     bHomed         :BOOL; 
     Pos_Done       :BOOL;   //定位完成
     Home_Alm      :BOOL;  //回零超时报警
     Pos_Alm         :BOOL; //定位超时报警



END_STRUCT
END_TYPE

// ---- P2DUTs/01_AxisCO_Ntrol/ST_JXCE.TcDUT
TYPE ST_JXCE :
STRUCT
      out_Control             AT  %Q*  :     UINT;  // 电机控制
      out_Function            AT  %Q*  :    UINT;  // 电机功能
      out_Start                 AT  %Q*  :   USINT;  // 电机启动定位
      out_Mode               AT  %Q*  :   USINT;  // 电机定位模式
      out_Cmd_Vel           AT  %Q*  :    UINT;  // 电机命令速度
      out_Cmd_Pos           AT  %Q*  :   DINT;  // 电机命令位置
      out_Cmd_Acc           AT  %Q*  :   UINT;  // 电机命令加速度
      out_Cmd_Dec          AT  %Q*  :    UINT;  // 电机命令减速度

      in_Status               AT  %I*  :     UINT;  // 电机状态
      in_Flag                 AT  %I*  :     UINT;  // 电机标志位
      in_Act_Pos              AT  %I*  :     DINT;  // 电机反馈位置
      in_Act_Vel             AT  %I*  :     UINT;  // 电机反馈速度
   
     in_Latest_Alm          AT  %I*  :     USINT;  // 电机最新报警

END_STRUCT
END_TYPE

// ---- P2DUTs/01_AxisCO_Ntrol/ST_SetpMotor.TcDUT
TYPE ST_SetpMotor :
STRUCT
	bJog_Up			:BOOL;		
	bJog_Down			:BOOL;	 
	bHome			:BOOL;	 
	bGoWorkPos			:BOOL;	 
	bLeaveWorkPos			:BOOL;	 
	HomeDone    :BOOL;  
	WorkPosDone :BOOL;
	
	
	
	biSensor  :BOOL;   //对射关电
	biUpSensor  :BOOL;   
	biRefSensor  :BOOL;   
	biMiddle2Sensor  :BOOL;   //步进中位感应 无用
	biDownSensor  :BOOL;  
	biBoxSensor  :BOOL;   //料盒到位感应
	bHave			:BOOL;//有料感应
	
	bo_Up			:BOOL;		
	bo_Down			:BOOL;	    

	bPoleFull: BOOL;  //极片料满

END_STRUCT
END_TYPE

// ---- P2DUTs/01_AxisCO_Ntrol_1/ST_AxisCmd.TcDUT
TYPE ST_AxisCmd :  //轴运动控制相关
STRUCT

   bDynamitcsParSel      :INT:=1;  // 1:NC          2:UserDefine


	bEnable			        :BOOL;				    (*使能*)
	fOverride			    :REAL:=100;			(*MC_power中实际倍率的设定，默认值为100*)
	bEnableFw		        :BOOL:=TRUE;		 (*正向使能*)
	bEnableBw		    :BOOL:=TRUE;	 	(*负向使能*)

	bJog_Fw			    :BOOL;			     	(*正向点动*)
	bJog_Bw			    :BOOL;			    	(*反向点动*)

	bMoveAbs	 	        :BOOL;				    (*运行绝对位置*)
	fPositon_of_Abs	 	:REAL;					(*绝对位置位移*)

	bMoveRel		        :BOOL;				   (*运行当对位置*)
	fPosition_of_Rel	    :REAL;				   (*相对位置位移*)

	bMoveModulo		 :BOOL;				     (*运行模长位置*)
	fPositon_of_Mod	  :REAL;					  (*模长位置位移*)

	bMoveVelo		    :BOOL;				       (*向一个方向持续运行，方向由前面的正向点动或者反向点动设置*)
	bMoveVeloDir	:MC_Direction := MC_Positive_Direction ;	(*速度运动的方向,MC_Negative_Direction*)

	bHome			       :BOOL;						(*启动回参*)

	bSetPos			       :BOOL;						 (*设置轴当前的位置为一个绝对位置*)
    fSetPos				   :REAL:=0;					(*setpos功能块将轴当前的位置设置为这个变量*)

	iGoSetPos              :INT;                     //GO离散点位_INT
    arrbGoSetPos      :ARRAY[0..15]        OF BOOL;  //GO离散点位_布尔数组
	iRealPoint              :INT;                     //离散点位指示_INIT
    arrbRealPoint        :ARRAY[0..15]        OF BOOL;  //离散点位指示_布尔数组

	bHalt			            :BOOL;				(*暂停*)
	bStop			        :BOOL;				(*停止*)
	bGearOut			    :BOOL;				(*解耦*)
	bReset			        :BOOL;				(*复位*)

	hmiJog_Fw			    :BOOL;				//正向点动_BOOL
	hmibJog_Bw		     :BOOL;				//反向点动_BOOL	
	hmiGoSetPos          :INT;              //GO离散点位_INT


//条件
     Home_Condition       :BOOL:=TRUE;//回原点条件
     JogP_Condition       :BOOL:=TRUE;//点动正转条件
     JogN_Condition       :BOOL:=TRUE;//点动反转条件
     GoPoint_Condition    :ARRAY[0..15] OF BOOL;//HMI点动定位条件


//轴到位判断
	Axis_R:REAL:=0.13;//轴到位判断





END_STRUCT
END_TYPE

// ---- P2DUTs/01_AxisCO_Ntrol_1/ST_AxisCtrl.TcDUT
TYPE ST_AxisCtrl :
STRUCT
    Io                        :ST_AxisIo;  (*轴IO信号*)
    Status                  :ST_AxisStatus;  
    Cmd                    :ST_AxisCmd;  
END_STRUCT
END_TYPE

// ---- P2DUTs/01_AxisCO_Ntrol_1/ST_AxisIo.TcDUT
TYPE ST_AxisIo :   //轴IO信号
STRUCT

	biNegLimit	             :BOOL;		            (*负限位触发信号*)
	biPosLimit	             :BOOL;		            (*正限位触发信号*)
	biHomeSwitch	     :BOOL;		         (*原点触发信号*)
    DigitalInputs          AT %I*	:  UDINT;
	
END_STRUCT
END_TYPE

// ---- P2DUTs/01_AxisCO_Ntrol_1/ST_AxisStatus.TcDUT
TYPE ST_AxisStatus :   //轴相关状态
STRUCT

(*status*)
	AxisName		     :STRING(31);		     (*轴名称*)
	AxisID			     :UDINT;		      (*轴在NC中的编号*)
	
    Enabled		         :BOOL;              //使能状态
	Moving              :BOOL;                //轴运行中
	NoMoving          :BOOL;   //轴停止中
    Coupled             :BOOL;   //轴耦合中

	fActPos			     :LREAL;  //轴的当前位置               
	fSetPos			     :LREAL;   //轴的指令位置              
    fModuloActPos		 :REAL;   //轴的当前模长位置             
    fModuloSetPos		 :REAL;      //轴的指令模长位置 
    fActVelo			   :REAL;    //轴的当前速度             
    fSetVelo			   :REAL;    //轴的指令速度
	Homed                :BOOL;        //轴回原点完成         
 
	Error                   :BOOL;//轴报错
	ErrorID                  :UDINT;//轴报错ID号
    WarningDynamitcsPar    :BOOL; //运动参数警告

     ErrorLimitSwitch           :BOOL; //限位报警
	 Errorcomp                   :BOOL; //手自动报警
END_STRUCT
END_TYPE

// ---- P2DUTs/01_AxisCO_Ntrol_1/ST_Axis_Par.TcDUT
TYPE ST_Axis_Par ://轴参数
STRUCT
    bLimitSwitchEn          :BOOL;//限位保护开启


	fVelocity_of_Abs	 :REAL:=5;				
	fVelocity_of_Mod	 :REAL:=5;				
	fVelocity_of_Rel	 :REAL:=5;				
	fVelocity_of_Velo	 :REAL:=5;				
	fVelocity_of_Jog	 :REAL:=10;			
	fInchingDistance	 :REAL:=5;				

	arrTargetPoint : ARRAY [0..15] OF REAL ;
	//fMaxVelocity:        REAL:=0;	
    fTagatTime                                 :REAL:=0.5;//S
    fConVelPercentage                      :REAL:=0.8;//S
    fMaxAccDec                              :LREAL:=40000;//最大加速度
    fMaxVel                                   :LREAL:=2000;//最大速度

	bHomeDirection                   :BOOL:=TRUE;
	fHomePosition                     :REAL:=10 ;	                          
	fHomeFastSpeed                  :REAL:=20 ;	 
	fHomeSlowSpeed                 :REAL:=10;	 
    HomeLimitDis                       :REAL:=5;	 

END_STRUCT
END_TYPE

// ---- P2DUTs/02_Cylinder/ST_CyCmd.TcDUT
TYPE ST_CyCmd ://
STRUCT
	bON:				        BOOL;	//开关ON
	bOFF:				    BOOL;	//开关OFF
	bFree:				    BOOL;	//泄压

    iType	:	                INT:=1	;	      //气缸类型选择：    1：气缸双控    2：气缸单控        3 电磁阀双控   4 电磁阀单控 
  
	OnCondition:		   BOOL:=TRUE;	//开条件
	OffCondition:		    BOOL:=TRUE;	//关条件
    ErrorTime:		        INT:=5;	

	HMION:	           BOOL;//HMI ON
	HMIOFF:	           BOOL;//HMI OFF


END_STRUCT
END_TYPE

// ---- P2DUTs/02_Cylinder/ST_CyCtrl.TcDUT
TYPE ST_CyCtrl ://气缸控制UDT  对应单控  双控气缸
STRUCT
   Io           : ST_CYIO;    //气缸IO
   Cmd      :  ST_CyCmd;
   Status     :ST_CyStatus;

END_STRUCT
END_TYPE

// ---- P2DUTs/02_Cylinder/ST_CYIo.TcDUT
TYPE ST_CYIo ://气缸 I O
STRUCT
	DIOnSwitch:		    BOOL;	//开限位
	DIOFFSwitch:		BOOL;	//关限位

	DOStatus1:          BOOL;//输出状态
	DOStatus2:          BOOL;//输出状态

END_STRUCT
END_TYPE

// ---- P2DUTs/02_Cylinder/ST_CyStatus.TcDUT
TYPE ST_CyStatus ://
STRUCT
	ONState:	        BOOL;//开状态
	OFFState:	        BOOL;//关状态
	Error1:	            BOOL;//气缸ON报警
	Error2:	            BOOL;//气缸OFF报警
    Errorcomp                   :BOOL; //手自动对 比报警
END_STRUCT
END_TYPE

// ---- P2DUTs/06_Interface/FB_Interface/ST_Cam.TcDUT
TYPE ST_Cam :  //张力FB 接口信号
STRUCT
   	bCamInExecute			                 :BOOL;	
   	bCreatTable		                         :BOOL;	

    bCreatTableDone                        :BOOL;
    bCreatTableError                        :BOOL;
	bError                                       :BOOL;

	bReady                                      :BOOL;
	bStartSync		                             :BOOL;
	bInSync		                                 :BOOL;//同步状态

END_STRUCT
END_TYPE

// ---- P2DUTs/06_Interface/FB_Interface/ST_Gear.TcDUT
TYPE ST_Gear : //
STRUCT
	bEnable		                        :BOOL;	
	bGearOutMode                 :BOOL;
 
	bReady                            :BOOL;  
	bInGear		 	                   :BOOL;	
	bError				               :BOOL;			
END_STRUCT
END_TYPE

// ---- P2DUTs/06_Interface/FB_Interface/ST_GearInPos.TcDUT
TYPE ST_GearInPos : //
STRUCT
	bEnable		                        :BOOL;	
   	bEnable2                       :BOOL;	

	bGearOutMode                 :BOOL;
    fMasterSyncPosition           :LREAL;  
    fSlaveSyncPosition              :LREAL;  

	bReady                            :BOOL;  
    bStartSync		 	               :BOOL;	
	bInSync		 	                   :BOOL;	
    bBusy                               :BOOL;	
	bError				               :BOOL;		

END_STRUCT
END_TYPE

// ---- P2DUTs/06_Interface/FB_Interface/ST_Tension.TcDUT
TYPE ST_Tension :  //张力FB 接口信号
STRUCT
	fWindDiameter           :REAL:=20;
    fDanserDegree           :REAL;
   
   	bTenExecute		        :BOOL;	
	bStudyExecute           :BOOL;       
   	fStudyDiameter          :REAL;  
	
	bReady                    :BOOL;  
	bTensionOK		       :BOOL;	

	bError			           :BOOL;	
                         
END_STRUCT
END_TYPE

// ---- P2DUTs/06_Interface/IData.TcDUT
TYPE IData :
STRUCT
	strBetryName:STRING;//CCD给电芯名称 
	bNGOverHang :BOOL;  //
	bHaveBetry :BOOL;   //当前工位是否有电芯
    
	
	bNGShort:BOOL;  //短路NG
	strShortData:STRING; //短路测试数据
	
	strCode:STRING;//二维码
    bNGCode:BOOL;   //二维码NG
	
	strHotPress:STRING;//热压参数
END_STRUCT
END_TYPE

// ---- P2DUTs/06_Interface/IM2Glue.TcDUT
TYPE IM2Glue :  //备胶方法st
STRUCT
    Start1:BOOL;   //备胶启动
	Done1:BOOL;   //备胶完成
	bActioning:BOOL;//备胶动作中	
	bAction2ing:BOOL;//贴胶动作中	

	Start2:BOOL;   //贴胶启
	iTagetPos : INT;  //贴胶位置
    Done2:BOOL;  //贴胶动作完成
	

	Reset:BOOL;  //复位
	AutoRuning:BOOL;  //运行中信号

END_STRUCT
END_TYPE

// ---- P2DUTs/06_Interface/Method/ST_Method.TcDUT
TYPE ST_Method :  //    方法
STRUCT

             AllTempTurnON                            :ST_MethodOut;//温控开

END_STRUCT
END_TYPE

// ---- P2DUTs/06_Interface/Method/ST_MethodOut.TcDUT
TYPE ST_MethodOut :  //    方法
STRUCT
             Execute            :BOOL;  
             Done1               :BOOL;  
             Done2               :BOOL;  
             Error               :BOOL;

END_STRUCT
END_TYPE

// ---- P2DUTs/07_Name/ST_Dust.TcDUT
TYPE ST_Dust :
STRUCT
FeedbeltDust1 :INT:=1;//负极送料皮带毛刷1
FeedbeltDust2 :INT:=2;//负极送料皮带毛刷2
FeedbeltDust3 :INT:=3;//负极送料皮带毛刷3
END_STRUCT
END_TYPE

// ---- P2DUTs/07_Name/ST_AxisName.TcDUT
TYPE ST_AxisName :
STRUCT
	AnCarryingLine	:INT;	//	正极送片搬运平移  1：取片位    2：放片位
	AnCarryingUpDown	:INT;	//	正极送片搬运升降 1：安全高度  2：取片高度	3：放片高度		4：等待高度
	AnCarryingWhirling	:INT;	//	正极送片搬运旋转	1：取片角度		2：放片角度
	AnDTCarryingLine	:INT;	//	正极叠台搬运平移1	1：取片位	2：放片位
	AnDTCarryingUpDown	:INT;	//	正极叠台搬运升降	1：安全高度		2：取片高度		3：放片高度		4：等待高度
	AndeviationX1	:INT;	//	正极纠偏平台X1持	1：初始位	2：纠偏位	3：标定位
	AndeviationX2	:INT;	//	正极纠偏平台X2	1：初始位	2：纠偏位	3：标定位
	AndeviationY	:INT;	//	正极纠偏平台Y		1：初始位	2：纠偏位	3：标定位
	CaCarryingLine1	:INT;	//	负极送片搬运1平移 		1：取片位	2：放片位
	CaCarryingUpDown1	:INT;	//	负极送片搬运1升降	1：安全高度		2：取片高度		3：放片高度		
	CaCarryingWhirling1	:INT;	//	负极送片搬运1旋转 	1：取片角度		2：放片角度
	CaCarryingLine2	:INT;	//	负极送片搬运2平移		1：取片位	2：放片位
	CaCarryingUpDown2	:INT;	//	负极送片搬运2升降	1：安全高度		2：取片高度		3：放片高度		4：等待高度
	CaBelt	:INT;	//	负极送片皮带
	CaDTCarryingLine	:INT;	//	负极叠台搬运平移	1：取片位  	2：放片位
	CaDTCarryingUpDown	:INT;	//	负极叠台搬运升降 	1：安全高度		2：取片高度		3：放片高度		4：等待高度 	5:避让高度
	CadeviationX1	:INT;	//	负极纠偏平台X1	1：初始位	2：纠偏位	3：标定位
	CadeviationX2	:INT;	//	负极纠偏平台X2 	1：初始位	2：纠偏位	3：标定位
	CadeviationY	:INT;	//	负极纠偏平台Y		1：初始位	2：纠偏位	3：标定位
	SEPTAunwinding	:INT;	//	隔膜放卷
	SEPTAdeviation1	:INT;	//	隔膜放卷纠偏	1：初始位
	SEPTAdeviation2	:INT;	//	隔膜尾部纠偏	1：初始位
	SEPTATension	:INT;	//	隔膜摆杆张力
	SEPTATCache	:INT;	//	隔膜缓存	1：初始位
	SEPTATLine	:INT;	//	隔膜平移	1：正极片位		2：负极片位
	DTUpDown	:INT;	//	叠台升降
	LeftYDLine	:INT;	//	左压刀开合	1：压紧位		2：张开位
	LeftYDUpDown	:INT;	//	左压刀升降 	1：初始位 11:张开高度 12：抽刀高度 13：过压高度 14：张开高度-过压高度 15：抽刀高度-过压高度 4:下料抽刀位 5：下料张开位
	RightYDLine	:INT;	//	右压刀开合 	1：压紧位		2：张开位
	RightYDUpDown	:INT;	//	右压刀升降 1：初始位 11:张开高度 12：抽刀高度 13：过压高度 14：张开高度-过压高度 15：抽刀高度-过压高度 4:下料抽刀位 5：下料张开位
	TailCurlLine	:INT;	//	尾卷夹电芯平移  	1：初始位（在初始位可旋转）	2：取电芯位 3：拉膜位	 4：尾卷位  5：尾卷避让位	6：下电芯位  7:回拉膜位 8:纠偏安全位 9：不尾卷切膜位 10:尾卷下料避让位 11:取电芯等待位
	TailCurlUpDown	:INT;	//	尾卷夹电芯升降   1：取电芯高度		2：夹膜高度		3：下电芯高度  4、放电芯下降位 5、尾卷高度 6、取对齐度NG料高度（变化要计算）7:尾卷完取料高度
	TailCurlRetracting	:INT;	//	尾卷夹电芯伸缩  1：初始位		2：取电芯位 		3：下电芯位
	TailCurlWhirling	:INT;	//	尾卷夹电芯旋转	1：取电芯位 	2：下电芯位	3:取电芯补偿位	4：取NG电芯补偿位
	TailCurlSEPTALine	:INT;	//	夹膜平移  1：初始位	 2:取电芯位	 3:夹膜平移原点到夹电芯平移原点距离 4:尾卷正常解耦位
	TailCurlSEPTAUpDown	:INT;	//	夹膜升降 1：取电芯高度 	2：夹膜高度 3:取对齐度NG料高度（变化要计算）
	LCurlingneedleLine	:INT;	//	长卷针平移	1：初始位	2：夹电芯位	3:尾卷补偿位1	4：尾卷补偿位2
	SCurlingneedleLine	:INT;	//	短卷针平移 	1：初始位	2：夹电芯位	
	LCurlingneedleWhirling	:INT;	//	长卷针旋转 1：初始位
	SCurlingneedleWhirling	:INT;	//	短卷针旋转	1：初始位
	
	GluingLine	:INT;	//	侧贴夹平移	1：左短边贴胶位1  2：左短边贴胶位2  3：右短边贴胶位1   4： 右短边贴胶位2  5:非极耳侧长边贴胶位 6:极耳侧长边贴胶位 8:上电芯位  9：下电芯位 10:尾卷安全旋转位
	GluingWhirling	:INT;	//	侧贴夹旋转   1：左短边贴胶位 2：右短边贴胶位  3：非极耳长边贴胶位  4：极耳长边贴胶位5:上电芯位   6:下电芯位
	GluingRetracting	:INT;	//	贴胶头进退  1:初始位   2：左短边贴胶位  3：右短边贴胶位   4：非极耳侧长边贴胶位  5：极耳侧长边贴胶位 6：踢NG胶位
	GluingUpDown	:INT;	//	拉胶升降 1： 拉二维胶初始位  2：拉二维胶切断位	3:二维胶取胶滚胶位 4：二维胶切胶滚胶位 5：拉蓝胶初始位 6：拉蓝胶切断位 7:蓝胶取胶滚胶位 8：蓝胶切胶滚胶位 9：踢废胶避让位
	
	Standby1	:INT;	//	备用
	Standby2	:INT;	//	备用		
END_STRUCT
END_TYPE

// ---- P2DUTs/07_Name/ST_CylinderName.TcDUT
TYPE ST_CylinderName :
STRUCT
AnScrapbinCy	:INT;		//		正极片NG收纳盒
CaScrapbinCy	:INT;		//		负极片NG收纳盒
CaScrapbinUDCy	:INT;		//		负极片NG收纳盒升降
PoleInflationCy	:INT;		//		隔膜放卷气胀轴
PoleTapeSplicerLCy	:INT;		//		隔膜接带左压板气缸
PoleTapeSplicerRCy	:INT;		//		隔膜接带右压板气缸
PreDiaph:INT;//叠台压隔膜气缸

PoleTapeCy	:INT;		//		隔膜夹紧气缸
PoleHotCutterCy	:INT;		//		隔膜热切升降
PoleSplintCy_U	:INT;		//		夹膜上夹板
PoleSplintCy_D	:INT;		//		夹膜下夹板


TailCurlSplintCy	:INT;		//		尾卷夹爪开合
CurlingSplintCy_L	:INT;		//		长卷针夹开合
CurlingSplintCy_S	:INT;		//		短卷针夹开合
CurlingSplintCy_S_1	:INT;		//		短卷针夹开合_1
TailCurlLineCy	:INT;		//		尾卷压辊平移缸
TailCurlUpdownCy	:INT;		//		尾卷压辊升降缸

StandbyGlueCy	:INT;		//		备蓝胶气缸
CodeStandbyGlueCy	:INT;		//		备二维码胶气缸

GlueClampsCy	:INT;		//		贴胶夹爪气缸

GluePressCy	:INT;		//		压蓝胶气缸
CodeGluePressCy	:INT;		//		压二维码胶气缸

GlueCutCy	:INT;		//		切蓝胶气缸
codeGlueCutCy	:INT;		//		切二维码胶气缸

PullGluePoleCy	:INT;		//		拉胶杆抱紧
PullGlueCy	:INT;		//		拉胶气缸
GlueNGCy	:INT;		//		踢废胶气缸
PullGlueModelCy	:INT;		//		贴胶治具托极耳

RollPoleearCy	:INT;		//尾卷托极耳托极耳

END_STRUCT
END_TYPE

// ---- P2DUTs/07_Name/ST_ElectValveName.TcDUT
TYPE ST_ElectValveName :
STRUCT
AnBeltVacuum	:INT;		//		正极模切送料分段皮带1取料处真空
AnBeltVacuumBark	:INT;		//		正极模切送料分段皮带1取料处破真空
CaMQBeltVacuum	:INT;		//		负极模切送料分段皮带1取料处真空
CaMQBeltVacuumBark	:INT;		//		负极模切送料分段皮带1取料处破真空
AnCarryingVacuum	:INT;		//		正极送片搬运升降真空
AnCarryingVacuumBark	:INT;		//		正极送片搬运升降破真空
AndeviationVacuum	:INT;		//		正极纠偏平台真空
AndeviationIonizedWind	:INT;		//		正极纠偏平台除尘风刀
AndeviationVacuumBark	:INT;		//		正极纠偏平台破真空
AnDTCarryingVacuum	:INT;		//		正极叠片搬运升降真空
AnDTCarryingJRVacuum	:INT;		//	正极叠片搬运升降极耳真空---ON有输出时破真空，没有输出时开真空
AnDTCarryingVacuumBark	:INT;		//		正极叠片搬运升降破真空
CaCarryingVacuum1	:INT;		//		负极送片搬运升降1真空
CaCarryingVacuumBark1	:INT;		//		负极送片搬运升降1破真空
CaLoadUpBeltVacuum	:INT;		//		负极送片皮带末端真空
CaLoadUpBeltVacuumBark	:INT;		//		负极送片皮带末端破真空
CaCarryingVacuum2	:INT;		//		负极送片搬运升降2真空---ON有输出时破真空，没有输出时开真空
CaCarryingVacuumBark2	:INT;		//		负极送片搬运升降2破真空
CadeviationVacuum	:INT;		//		负极纠偏平台真空
CadeviationVacuumBark	:INT;		//		负极纠偏平台破真空
CadeviationIonizedWind	:INT;		//		负极纠偏平台除尘风刀
CaDTCarryingVacuum	:INT;		//		负极叠片搬运升降真空---ON有输出时破真空，没有输出时开真空
CaDTCarryingJRVacuum	:INT;		//	负极叠片搬运升降极耳真空---ON有输出时破真空，没有输出时开真空
CaDTCarryingVacuumBark	:INT;		//		负极叠片搬运升降破真空
PoleTapeDustRemoval	:INT;		//		隔膜接带平台除尘
PoleTapeVacuum	:INT;		//		隔膜接带平台真空
BlueGlueVacuum1	:INT;		//		备胶组件蓝胶真空1
BlueGlueVacuum2	:INT;		//		备胶组件蓝胶真空2
codeGlueVacuum1	:INT;		//		备胶组件二维码胶真空1
codeGlueVacuum2	:INT;		//		备胶组件二维码胶真空2
PastesGlueVacuum	:INT;		//		备胶组件贴胶头真空
DTVacuum	:INT;		//		叠片台真空
PoleSplintVacuum_D	:INT;		//		夹膜下夹板真空
WJ_blow:INT;//尾卷夹电芯吹气
WJShortvacuum:INT;//短卷针张开真空
END_STRUCT
END_TYPE

// ---- P2DUTs/07_Name/ST_P2AxisName.TcDUT
TYPE ST_P2AxisName :   //2#部分轴
STRUCT
P2M1_AnCarryingLine	:INT:=1;	//1号叠台	正极送片搬运平移 
P2M1_AnCarryingUpDown	:INT:=2;	//1号叠台	正极送片搬运升降
P2M1_AnCarryingWhirling	:INT:=3;	//1号叠台	正极送片搬运旋转
P2M1_AnDTCarryingLine	:INT:=4;	//1号叠台	正极叠台搬运平移1
P2M1_AnDTCarryingUpDown	:INT:=5;	//1号叠台	正极叠台搬运升降
P2M1_AndeviationX1	:INT:=6;	//1号叠台	正极纠偏平台X1
P2M1_AndeviationX2	:INT:=7;	//1号叠台	正极纠偏平台X2
P2M1_AndeviationY	:INT:=8;	//1号叠台	正极纠偏平台Y
P2M1_CaCarryingLine1	:INT:=9;	//1号叠台	负极送片搬运1平移
P2M1_CaCarryingUpDown1	:INT:=10;	//1号叠台	负极送片搬运1升降
P2M1_CaCarryingWhirling1	:INT:=11;	//1号叠台	负极送片搬运1旋转
P2M1_CaCarryingLine2	:INT:=12;	//1号叠台	负极送片搬运2平移
P2M1_CaCarryingUpDown2	:INT:=13;	//1号叠台	负极送片搬运2升降
P2M1_CaBelt	:INT:=14;	//1号叠台	负极送片皮带
P2M1_CaDTCarryingLine	:INT:=15;	//1号叠台	负极叠台搬运平移
P2M1_CaDTCarryingUpDown	:INT:=16;	//1号叠台	负极叠台搬运升降
P2M1_CadeviationX1	:INT:=17;	//1号叠台	负极纠偏平台X1
P2M1_CadeviationX2	:INT:=18;	//1号叠台	负极纠偏平台X2
P2M1_CadeviationY	:INT:=19;	//1号叠台	负极纠偏平台Y
P2M1_SEPTAunwinding	:INT:=20;	//1号叠台	隔膜放卷
P2M1_SEPTAdeviation1	:INT:=21;	//1号叠台	隔膜放卷纠偏
P2M1_SEPTAdeviation2	:INT:=22;	//1号叠台	隔膜尾部纠偏
P2M1_SEPTATension	:INT:=23;	//1号叠台	隔膜摆杆张力
P2M1_SEPTATCache	:INT:=24;	//1号叠台	隔膜缓存
P2M1_SEPTATLine	:INT:=25;	//1号叠台	隔膜平移
P2M1_DTUpDown	:INT:=26;	//1号叠台	叠台升降
P2M1_LeftYDLine	:INT:=27;	//1号叠台	左压刀开合
P2M1_LeftYDUpDown	:INT:=28;	//1号叠台	左压刀升降
P2M1_RightYDLine	:INT:=29;	//1号叠台	右压刀开合
P2M1_RightYDUpDown	:INT:=30;	//1号叠台	右压刀升降
P2M1_TailCurlLine	:INT:=31;	//1号叠台	尾卷夹电芯平移
P2M1_TailCurlUpDown	:INT:=32;	//1号叠台	尾卷夹电芯升降
P2M1_TailCurlRetracting	:INT:=33;	//1号叠台	尾卷夹电芯伸缩
P2M1_TailCurlWhirling	:INT:=34;	//1号叠台	尾卷夹电芯旋转
P2M1_TailCurlSEPTALine	:INT:=35;	//1号叠台	夹膜平移
P2M1_TailCurlSEPTAUpDown	:INT:=36;	//1号叠台	夹膜升降
P2M1_LCurlingneedleLine	:INT:=37;	//1号叠台	长卷针平移
P2M1_SCurlingneedleLine	:INT:=38;	//1号叠台	短卷针平移
P2M1_LCurlingneedleWhirling	:INT:=39;	//1号叠台	长卷针旋转
P2M1_SCurlingneedleWhirling	:INT:=40;	//1号叠台	短卷针旋转
P2M1_GluingLine	:INT:=41;	//1号叠台	侧贴夹平移
P2M1_GluingWhirling	:INT:=42;	//1号叠台	侧贴夹旋转
P2M1_GluingRetracting	:INT:=43;	//1号叠台	贴胶头进退
P2M1_GluingUpDown	:INT:=44;	//1号叠台	拉胶升降
P2M1_Standby1	:INT:=45;	//1号叠台	备用
P2M1_Standby2	:INT:=46;	//1号叠台	备用

P2M2_AnCarryingLine	:INT:=47;	//2号叠台	正极送片搬运平移
P2M2_AnCarryingUpDown	:INT:=48;	//2号叠台	正极送片搬运升降
P2M2_AnCarryingWhirling	:INT:=49;	//2号叠台	正极送片搬运旋转
P2M2_AnDTCarryingLine	:INT:=50;	//2号叠台	正极叠台搬运平移
P2M2_AnDTCarryingUpDown	:INT:=51;	//2号叠台	正极叠台搬运升降
P2M2_AndeviationX1	:INT:=52;	//2号叠台	正极纠偏平台X1
P2M2_AndeviationX2	:INT:=53;	//2号叠台	正极纠偏平台X2
P2M2_AndeviationY	:INT:=54;	//2号叠台	正极纠偏平台Y
P2M2_CaCarryingLine1	:INT:=55;	//2号叠台	负极送片搬运1平移
P2M2_CaCarryingUpDown1	:INT:=56;	//2号叠台	负极送片搬运1升降
P2M2_CaCarryingWhirling1	:INT:=57;	//2号叠台	负极送片搬运1旋转
P2M2_CaCarryingLine2	:INT:=58;	//2号叠台	负极送片搬运2平移
P2M2_CaCarryingUpDown2	:INT:=59;	//2号叠台	负极送片搬运2升降
P2M2_CaBelt	:INT:=60;	//2号叠台	负极送片皮带
P2M2_CaDTCarryingLine	:INT:=61;	//2号叠台	负极叠台搬运平移
P2M2_CaDTCarryingUpDown	:INT:=62;	//2号叠台	负极叠台搬运升降
P2M2_CadeviationX1	:INT:=63;	//2号叠台	负极纠偏平台X1
P2M2_CadeviationX2	:INT:=64;	//2号叠台	负极纠偏平台X2
P2M2_CadeviationY	:INT:=65;	//2号叠台	负极纠偏平台Y
P2M2_SEPTAunwinding	:INT:=66;	//2号叠台	隔膜放卷
P2M2_SEPTAdeviation1	:INT:=67;	//2号叠台	隔膜放卷纠偏
P2M2_SEPTAdeviation2	:INT:=68;	//2号叠台	隔膜尾部纠偏
P2M2_SEPTATension	:INT:=69;	//2号叠台	隔膜摆杆张力
P2M2_SEPTATCache	:INT:=70;	//2号叠台	隔膜缓存
P2M2_SEPTATLine	:INT:=71;	//2号叠台	隔膜平移
P2M2_DTUpDown	:INT:=72;	//2号叠台	叠台升降
P2M2_LeftYDLine	:INT:=73;	//2号叠台	左压刀开合
P2M2_LeftYDUpDown	:INT:=74;	//2号叠台	左压刀升降
P2M2_RightYDLine	:INT:=75;	//2号叠台	右压刀开合
P2M2_RightYDUpDown	:INT:=76;	//2号叠台	右压刀升降
P2M2_TailCurlLine	:INT:=77;	//2号叠台	尾卷夹电芯平移
P2M2_TailCurlUpDown	:INT:=78;	//2号叠台	尾卷夹电芯升降
P2M2_TailCurlRetracting	:INT:=79;	//2号叠台	尾卷夹电芯伸缩
P2M2_TailCurlWhirling	:INT:=80;	//2号叠台	尾卷夹电芯旋转
P2M2_TailCurlSEPTALine	:INT:=81;	//2号叠台	夹膜平移
P2M2_TailCurlSEPTAUpDown	:INT:=82;	//2号叠台	夹膜升降
P2M2_LCurlingneedleLine	:INT:=83;	//2号叠台	长卷针平移
P2M2_SCurlingneedleLine	:INT:=84;	//2号叠台	短卷针平移
P2M2_LCurlingneedleWhirling	:INT:=85;	//2号叠台	长卷针旋转
P2M2_SCurlingneedleWhirling	:INT:=86;	//2号叠台	短卷针旋转
P2M2_GluingLine	:INT:=87;	//2号叠台	侧贴夹平移
P2M2_GluingWhirling	:INT:=88;	//2号叠台	侧贴夹旋转
P2M2_GluingRetracting	:INT:=89;	//2号叠台	贴胶头进退
P2M2_GluingUpDown	:INT:=90;	//2号叠台	拉胶升降
P2M2_Standby1	:INT:=91;	//2号叠台	备用
P2M2_Standby2	:INT:=92;	//2号叠台	备用

P2M3_AnCarryingLine	:INT:=93;	//3号叠台	正极送片搬运平移
P2M3_AnCarryingUpDown	:INT:=94;	//3号叠台	正极送片搬运升降
P2M3_AnCarryingWhirling	:INT:=95;	//3号叠台	正极送片搬运旋转
P2M3_AnDTCarryingLine	:INT:=96;	//3号叠台	正极叠台搬运平移
P2M3_AnDTCarryingUpDown	:INT:=97;	//3号叠台	正极叠台搬运升降
P2M3_AndeviationX1	:INT:=98;	//3号叠台	正极纠偏平台X1
P2M3_AndeviationX2	:INT:=99;	//3号叠台	正极纠偏平台X2
P2M3_AndeviationY	:INT:=100;	//3号叠台	正极纠偏平台Y
P2M3_CaCarryingLine1	:INT:=101;	//3号叠台	负极送片搬运1平移
P2M3_CaCarryingUpDown1	:INT:=102;	//3号叠台	负极送片搬运1升降
P2M3_CaCarryingWhirling1	:INT:=103;	//3号叠台	负极送片搬运1旋转
P2M3_CaCarryingLine2	:INT:=104;	//3号叠台	负极送片搬运2平移
P2M3_CaCarryingUpDown2	:INT:=105;	//3号叠台	负极送片搬运2升降
P2M3_CaBelt	:INT:=106;	//3号叠台	负极送片皮带
P2M3_CaDTCarryingLine	:INT:=107;	//3号叠台	负极叠台搬运平移
P2M3_CaDTCarryingUpDown	:INT:=108;	//3号叠台	负极叠台搬运升降
P2M3_CadeviationX1	:INT:=109;	//3号叠台	负极纠偏平台X1
P2M3_CadeviationX2	:INT:=110;	//3号叠台	负极纠偏平台X2
P2M3_CadeviationY	:INT:=111;	//3号叠台	负极纠偏平台Y
P2M3_SEPTAunwinding	:INT:=112;	//3号叠台	隔膜放卷
P2M3_SEPTAdeviation1	:INT:=113;	//3号叠台	隔膜放卷纠偏
P2M3_SEPTAdeviation2	:INT:=114;	//3号叠台	隔膜尾部纠偏
P2M3_SEPTATension	:INT:=115;	//3号叠台	隔膜摆杆张力
P2M3_SEPTATCache	:INT:=116;	//3号叠台	隔膜缓存
P2M3_SEPTATLine	:INT:=117;	//3号叠台	隔膜平移
P2M3_DTUpDown	:INT:=118;	//3号叠台	叠台升降
P2M3_LeftYDLine	:INT:=119;	//3号叠台	左压刀开合
P2M3_LeftYDUpDown	:INT:=120;	//3号叠台	左压刀升降
P2M3_RightYDLine	:INT:=121;	//3号叠台	右压刀开合
P2M3_RightYDUpDown	:INT:=122;	//3号叠台	右压刀升降
P2M3_TailCurlLine	:INT:=123;	//3号叠台	尾卷夹电芯平移
P2M3_TailCurlUpDown	:INT:=124;	//3号叠台	尾卷夹电芯升降
P2M3_TailCurlRetracting	:INT:=125;	//3号叠台	尾卷夹电芯伸缩
P2M3_TailCurlWhirling	:INT:=126;	//3号叠台	尾卷夹电芯旋转
P2M3_TailCurlSEPTALine	:INT:=127;	//3号叠台	夹膜平移
P2M3_TailCurlSEPTAUpDown	:INT:=128;	//3号叠台	夹膜升降
P2M3_LCurlingneedleLine	:INT:=129;	//3号叠台	长卷针平移
P2M3_SCurlingneedleLine	:INT:=130;	//3号叠台	短卷针平移
P2M3_LCurlingneedleWhirling	:INT:=131;	//3号叠台	长卷针旋转
P2M3_SCurlingneedleWhirling	:INT:=132;	//3号叠台	短卷针旋转
P2M3_GluingLine	:INT:=133;	//3号叠台	侧贴夹平移
P2M3_GluingWhirling	:INT:=134;	//3号叠台	侧贴夹旋转
P2M3_GluingRetracting	:INT:=135;	//3号叠台	贴胶头进退
P2M3_GluingUpDown	:INT:=136;	//3号叠台	拉胶升降
P2M3_Standby1	:INT:=137;	//3号叠台	备用
P2M3_Standby2	:INT:=138;	//3号叠台	备用


END_STRUCT
END_TYPE

// ---- P2DUTs/07_Name/ST_P2CylinderName.TcDUT
TYPE ST_P2CylinderName :   //2#部分气缸
STRUCT
P2M1_AnScrapbinCy	:INT:=1;		//1号叠台		正极片NG收纳盒
P2M1_CaScrapbinCy	:INT:=2;		//1号叠台		负极片NG收纳盒
P2M1_CaScrapbinUDCy	:INT:=3;		//1号叠台		负极片NG收纳盒升降
P2M1_StackpreCy	:INT:=4;		//1号叠台		叠台压刀气缸
P2M1_PreDiaph	:INT:=5;		//1号叠台		压隔膜气缸
P2M1_PoleInflationCy	:INT:=6;		//1号叠台		隔膜放卷气胀轴
P2M1_PoleTapeSplicerLCy	:INT:=7;		//1号叠台		隔膜接带左压板气缸
P2M1_PoleTapeSplicerRCy	:INT:=8;		//1号叠台		隔膜接带右压板气缸
P2M1_PoleTapeCy	:INT:=9;		//1号叠台		隔膜夹紧气缸
P2M1_PoleHotCutterCy	:INT:=10;		//1号叠台		隔膜热切升降
P2M1_PoleSplintCy_U	:INT:=11;		//1号叠台		夹膜上夹板
P2M1_PoleSplintCy_D	:INT:=12;		//1号叠台		夹膜下夹板
P2M1_TailCurlSplintCy	:INT:=13;		//1号叠台		尾卷夹爪开合
P2M1_CurlingSplintCy_L	:INT:=14;		//1号叠台		长卷针夹开合
P2M1_CurlingSplintCy_S	:INT:=15;		//1号叠台		短卷针夹开合
P2M1_TailCurlLineCy	:INT:=16;		//1号叠台		尾卷压辊平移缸
P2M1_TailCurlUpdownCy	:INT:=17;		//1号叠台		尾卷压辊升降缸
P2M1_StandbyGlueCy	:INT:=18;		//1号叠台		备胶气缸
P2M1_CodeStandbyGlueCy	:INT:=19;		//1号叠台		备二维码胶气缸
P2M1_GlueClampsCy	:INT:=20;		//1号叠台		贴胶夹爪气缸
P2M1_GluePressCy	:INT:=21;		//1号叠台		压胶气缸
P2M1_CodeGluePressCy	:INT:=22;		//1号叠台		压二维码胶气缸
P2M1_GlueCutCy	:INT:=23;		//1号叠台		切胶气缸
P2M1_codeGlueCutCy	:INT:=24;		//1号叠台		切二维码胶气缸
P2M1_PullGluePoleCy	:INT:=25;		//1号叠台		拉胶杆抱紧
P2M1_PullGlueCy	:INT:=26;		//1号叠台		拉胶气缸
P2M1_GlueNGCy	:INT:=27;		//1号叠台		踢废胶气缸
P2M1_PullGlueModelCy	:INT:=28;		//1号叠台		贴胶治具气缸

P2M2_AnScrapbinCy	:INT:=29;		//2号叠台		正极片NG收纳盒
P2M2_CaScrapbinCy	:INT:=30;		//2号叠台		负极片NG收纳盒
P2M2_StackpreCy	:INT:=31;		//2号叠台		叠台压刀气缸
P2M2_PreDiaphCy	:INT:=32;		//2号叠台		压隔膜气缸
P2M2_PoleTapeCy	:INT:=33;		//2号叠台		隔膜夹紧气缸
P2M2_PoleInflationCy	:INT:=34;		//2号叠台		隔膜放卷气胀轴
P2M2_PoleTapeSplicerLCy	:INT:=35;		//2号叠台		隔膜接带左压板气缸
P2M2_PoleTapeSplicerRCy	:INT:=36;		//2号叠台		隔膜接带右压板气缸
P2M2_CaScrapbinUDCy	:INT:=37;		//2号叠台		负极片NG收纳盒升降
P2M2_PoleHotCutterCy	:INT:=38;		//2号叠台		隔膜热切升降
P2M2_PoleSplintCy_U	:INT:=39;		//2号叠台		夹膜上夹板
P2M2_PoleSplintCy_D	:INT:=40;		//2号叠台		夹膜下夹板
P2M2_TailCurlSplintCy	:INT:=41;		//2号叠台		尾卷夹爪开合
P2M2_CurlingSplintCy_L	:INT:=42;		//2号叠台		长卷针夹开合
P2M2_CurlingSplintCy_S	:INT:=43;		//2号叠台		短卷针夹开合
P2M2_TailCurlLineCy	:INT:=44;		//2号叠台		尾卷压辊平移缸
P2M2_TailCurlUpdownCy	:INT:=45;		//2号叠台		尾卷压辊升降缸
P2M2_StandbyGlueCy	:INT:=46;		//2号叠台		备胶气缸
P2M2_CodeStandbyGlueCy	:INT:=47;		//2号叠台		备二维码胶气缸
P2M2_GlueClampsCy	:INT:=48;		//2号叠台		贴胶夹爪气缸
P2M2_GluePressCy	:INT:=49;		//2号叠台		压胶气缸
P2M2_CodeGluePressCy	:INT:=50;		//2号叠台		压二维码胶气缸
P2M2_GlueCutCy	:INT:=51;		//2号叠台		切胶气缸
P2M2_codeGlueCutCy	:INT:=52;		//2号叠台		切二维码胶气缸
P2M2_PullGluePoleCy	:INT:=53;		//2号叠台		拉胶杆抱紧
P2M2_PullGlueCy	:INT:=54;		//2号叠台		拉胶气缸
P2M2_GlueNGCy	:INT:=55;		//2号叠台		踢废胶气缸
P2M2_PullGlueModelCy	:INT:=56;		//2号叠台		贴胶治具气缸

P2M3_AnScrapbinCy	:INT:=57;		//3号叠台		正极片NG收纳盒
P2M3_CaScrapbinCy	:INT:=58;		//3号叠台		负极片NG收纳盒
P2M3_CaScrapbinUDCy	:INT:=59;		//3号叠台		负极片NG收纳盒升降
P2M3_StackpreCy	:INT:=60;		//3号叠台		叠台压刀气缸
P2M3_PreDiaphCy	:INT:=61;		//3号叠台		压隔膜气缸
P2M3_PoleInflationCy	:INT:=62;		//3号叠台		隔膜放卷气胀轴
P2M3_PoleTapeSplicerLCy	:INT:=63;		//3号叠台		隔膜接带左压板气缸
P2M3_PoleTapeSplicerRCy	:INT:=64;		//3号叠台		隔膜接带右压板气缸
P2M3_PoleTapeCy	:INT:=65;		//3号叠台		隔膜夹紧气缸
P2M3_PoleHotCutterCy	:INT:=66;		//3号叠台		隔膜热切升降
P2M3_PoleSplintCy_U	:INT:=67;		//3号叠台		夹膜上夹板
P2M3_PoleSplintCy_D	:INT:=68;		//3号叠台		夹膜下夹板
P2M3_TailCurlSplintCy	:INT:=69;		//3号叠台		尾卷夹爪开合
P2M3_CurlingSplintCy_L	:INT:=70;		//3号叠台		长卷针夹开合
P2M3_CurlingSplintCy_S	:INT:=71;		//3号叠台		短卷针夹开合
P2M3_TailCurlLineCy	:INT:=72;		//3号叠台		尾卷压辊平移缸
P2M3_TailCurlUpdownCy	:INT:=73;		//3号叠台		尾卷压辊升降缸
P2M3_StandbyGlueCy	:INT:=74;		//3号叠台		备胶气缸
P2M3_CodeStandbyGlueCy	:INT:=75;		//3号叠台		备二维码胶气缸
P2M3_GlueClampsCy	:INT:=76;		//3号叠台		贴胶夹爪气缸
P2M3_GluePressCy	:INT:=77;		//3号叠台		压胶气缸
P2M3_CodeGluePressCy	:INT:=78;		//3号叠台		压二维码胶气缸
P2M3_GlueCutCy	:INT:=79;		//3号叠台		切胶气缸
P2M3_codeGlueCutCy	:INT:=80;		//3号叠台		切二维码胶气缸
P2M3_PullGluePoleCy	:INT:=81;		//3号叠台		拉胶杆抱紧
P2M3_PullGlueCy	:INT:=82;		//3号叠台		拉胶气缸
P2M3_GlueNGCy	:INT:=83;		//3号叠台		踢废胶气缸
P2M3_PullGlueModelCy	:INT:=84;		//3号叠台		贴胶治具气缸
LockonCy:INT:=85;//电芯NG1料盒锁定气缸
P2M3_CurlingSplintCy_S_1	:INT:=86;		//3号叠台		短卷针夹泄气
P2M2_CurlingSplintCy_S_1	:INT:=87;		//2号叠台		短卷针夹泄气
P2M1_CurlingSplintCy_S_1    :INT:=88;		//1号叠台		短卷针夹泄气

P2M1_RollPoleearCy    :INT:=89;		//1号叠台		尾卷托极耳气缸
P2M2_RollPoleearCy    :INT:=90;		//2号叠台		尾卷托极耳气缸
P2M3_RollPoleearCy    :INT:=91;		//3号叠台		尾卷托极耳气缸
END_STRUCT
END_TYPE

// ---- P2DUTs/07_Name/ST_P2ElectValveName.TcDUT
TYPE ST_P2ElectValveName :   //2#部分气缸
STRUCT
P2M1_AnBeltVacuum	:INT:=110;	//1号叠台		正极模切送料分段皮带1取料处真空
P2M1_AnBeltVacuumBark	:INT:=111;	//1号叠台		正极模切送料分段皮带1取料处破真空
P2M1_CaMQBeltVacuum	:INT:=112;	//1号叠台		负极模切送料分段皮带1取料处真空
P2M1_CaMQBeltVacuumBark	:INT:=113;	//1号叠台		负极模切送料分段皮带1取料处破真空
P2M1_AnCarryingVacuum	:INT:=114;	//1号叠台		正极送片搬运升降真空
P2M1_AnCarryingVacuumBark	:INT:=115;	//1号叠台		正极送片搬运升降破真空
P2M1_AndeviationVacuum	:INT:=116;	//1号叠台		正极纠偏平台真空
P2M1_AndeviationIonizedWind	:INT:=117;	//1号叠台		正极纠偏平台除尘风刀
P2M1_AndeviationVacuumBark	:INT:=118;	//1号叠台		正极纠偏平台破真空
P2M1_AnDTCarryingVacuum	:INT:=119;	//1号叠台		正极叠片搬运升降真空
P2M1_AnDTCarryingVacuumBark	:INT:=120;	//1号叠台		正极叠片搬运升降破真空
P2M1_CaCarryingVacuum1	:INT:=121;	//1号叠台		负极送片搬运升降1真空
P2M1_CaCarryingVacuumBark1	:INT:=122;	//1号叠台		负极送片搬运升降1破真空
P2M1_CaLoadUpBeltVacuum	:INT:=123;	//1号叠台		负极送片皮带末端真空
P2M1_CaLoadUpBeltVacuumBark	:INT:=124;	//1号叠台		负极送片皮带末端破真空
P2M1_CaCarryingVacuum2	:INT:=125;	//1号叠台		负极送片搬运升降2真空
P2M1_CaCarryingVacuumBark2	:INT:=126;	//1号叠台		负极送片搬运升降2破真空
P2M1_CadeviationVacuum	:INT:=127;	//1号叠台		负极纠偏平台真空
P2M1_CadeviationVacuumBark	:INT:=128;	//1号叠台		负极纠偏平台破真空
P2M1_CadeviationIonizedWind	:INT:=129;	//1号叠台		负极纠偏平台除尘风刀
P2M1_CaDTCarryingVacuum	:INT:=130;	//1号叠台		负极叠片搬运升降真空
P2M1_CaDTCarryingVacuumBark	:INT:=131;	//1号叠台		负极叠片搬运升降破真空
P2M1_PoleTapeDustRemoval	:INT:=132;	//1号叠台		隔膜接带平台除尘
P2M1_PoleTapeVacuum	:INT:=133;	//1号叠台		隔膜接带平台真空
P2M1_BlueGlueVacuum1	:INT:=134;	//1号叠台		备胶组件蓝胶真空1
P2M1_BlueGlueVacuum2	:INT:=135;	//1号叠台		备胶组件蓝胶真空2
P2M1_codeGlueVacuum1	:INT:=136;	//1号叠台		备胶组件二维码胶真空1
P2M1_codeGlueVacuum2	:INT:=137;	//1号叠台		备胶组件二维码胶真空2
P2M1_PastesGlueVacuum	:INT:=138;	//1号叠台		备胶组件贴胶头真空
P2M1_DTVacuum	:INT:=139;	//1号叠台		叠片台真空
P2M1_PoleSplintVacuum_D	:INT:=140;	//1号叠台		夹膜下夹板真空
P2M2_AnBeltVacuum	:INT:=141;	//2号叠台		正极模切送料分段皮带1取料处真空
P2M2_AnBeltVacuumBark	:INT:=142;	//2号叠台		正极模切送料分段皮带1取料处破真空
P2M2_CaMQBeltVacuum	:INT:=143;	//2号叠台		负极模切送料分段皮带1取料处真空
P2M2_CaMQBeltVacuumBark	:INT:=144;	//2号叠台		负极模切送料分段皮带1取料处破真空
P2M2_AnCarryingVacuum	:INT:=145;	//2号叠台		正极送片搬运升降真空
P2M2_AnCarryingVacuumBark	:INT:=146;	//2号叠台		正极送片搬运升降破真空
P2M2_AndeviationVacuum	:INT:=147;	//2号叠台		正极纠偏平台真空
P2M2_AndeviationIonizedWind	:INT:=148;	//2号叠台		正极纠偏平台除尘风刀
P2M2_AndeviationVacuumBark	:INT:=149;	//2号叠台		正极纠偏平台破真空
P2M2_AnDTCarryingVacuum	:INT:=150;	//2号叠台		正极叠片搬运升降真空
P2M2_AnDTCarryingVacuumBark	:INT:=151;	//2号叠台		正极叠片搬运升降破真空
P2M2_CaCarryingVacuum1	:INT:=152;	//2号叠台		负极送片搬运升降1真空
P2M2_CaCarryingVacuumBark1	:INT:=153;	//2号叠台		负极送片搬运升降1破真空
P2M2_CaLoadUpBeltVacuum	:INT:=154;	//2号叠台		负极送片皮带末端真空
P2M2_CaLoadUpBeltVacuumBark	:INT:=155;	//2号叠台		负极送片皮带末端破真空
P2M2_CaCarryingVacuum2	:INT:=156;	//2号叠台		负极送片搬运升降2真空
P2M2_CaCarryingVacuumBark2	:INT:=157;	//2号叠台		负极送片搬运升降2破真空
P2M2_CadeviationVacuum	:INT:=158;	//2号叠台		负极纠偏平台真空
P2M2_CadeviationVacuumBark	:INT:=159;	//2号叠台		负极纠偏平台破真空
P2M2_CadeviationIonizedWind	:INT:=160;	//2号叠台		负极纠偏平台除尘风刀
P2M2_CaDTCarryingVacuum	:INT:=161;	//2号叠台		负极叠片搬运升降真空
P2M2_CaDTCarryingVacuumBark	:INT:=162;	//2号叠台		负极叠片搬运升降破真空
P2M2_PoleTapeDustRemoval	:INT:=163;	//2号叠台		隔膜接带平台除尘
P2M2_PoleTapeVacuum	:INT:=164;	//2号叠台		隔膜接带平台真空
P2M2_BlueGlueVacuum1	:INT:=165;	//2号叠台		备胶组件蓝胶真空1
P2M2_BlueGlueVacuum2	:INT:=166;	//2号叠台		备胶组件蓝胶真空2
P2M2_codeGlueVacuum1	:INT:=167;	//2号叠台		备胶组件二维码胶真空1
P2M2_codeGlueVacuum2	:INT:=168;	//2号叠台		备胶组件二维码胶真空2
P2M2_PastesGlueVacuum	:INT:=169;	//2号叠台		备胶组件贴胶头真空
P2M2_DTVacuum	:INT:=170;	//2号叠台		叠片台真空
P2M2_PoleSplintVacuum_D	:INT:=171;	//2号叠台		夹膜下夹板真空
P2M3_AnBeltVacuum	:INT:=172;	//3号叠台		正极模切送料分段皮带1取料处真空
P2M3_AnBeltVacuumBark	:INT:=173;	//3号叠台		正极模切送料分段皮带1取料处破真空
P2M3_CaMQBeltVacuum	:INT:=174;	//3号叠台		负极模切送料分段皮带1取料处真空
P2M3_CaMQBeltVacuumBark	:INT:=175;	//3号叠台		负极模切送料分段皮带1取料处破真空
P2M3_AnCarryingVacuum	:INT:=176;	//3号叠台		正极送片搬运升降真空
P2M3_AnCarryingVacuumBark	:INT:=177;	//3号叠台		正极送片搬运升降破真空
P2M3_AndeviationVacuum	:INT:=178;	//3号叠台		正极纠偏平台真空
P2M3_AndeviationIonizedWind	:INT:=179;	//3号叠台		正极纠偏平台除尘风刀
P2M3_AndeviationVacuumBark	:INT:=180;	//3号叠台		正极纠偏平台破真空
P2M3_AnDTCarryingVacuum	:INT:=181;	//3号叠台		正极叠片搬运升降真空
P2M3_AnDTCarryingVacuumBark	:INT:=182;	//3号叠台		正极叠片搬运升降破真空
P2M3_CaCarryingVacuum1	:INT:=183;	//3号叠台		负极送片搬运升降1真空
P2M3_CaCarryingVacuumBark1	:INT:=184;	//3号叠台		负极送片搬运升降1破真空
P2M3_CaLoadUpBeltVacuum	:INT:=185;	//3号叠台		负极送片皮带末端真空
P2M3_CaLoadUpBeltVacuumBark	:INT:=186;	//3号叠台		负极送片皮带末端破真空
P2M3_CaCarryingVacuum2	:INT:=187;	//3号叠台		负极送片搬运升降2真空
P2M3_CaCarryingVacuumBark2	:INT:=188;	//3号叠台		负极送片搬运升降2破真空
P2M3_CadeviationVacuum	:INT:=189;	//3号叠台		负极纠偏平台真空
P2M3_CadeviationVacuumBark	:INT:=190;	//3号叠台		负极纠偏平台破真空
P2M3_CadeviationIonizedWind	:INT:=191;	//3号叠台		负极纠偏平台除尘风刀
P2M3_CaDTCarryingVacuum	:INT:=192;	//3号叠台		负极叠片搬运升降真空
P2M3_CaDTCarryingVacuumBark	:INT:=193;	//3号叠台		负极叠片搬运升降破真空
P2M3_PoleTapeDustRemoval	:INT:=194;	//3号叠台		隔膜接带平台除尘
P2M3_PoleTapeVacuum	:INT:=195;	//3号叠台		隔膜接带平台真空
P2M3_BlueGlueVacuum1	:INT:=196;	//3号叠台		备胶组件蓝胶真空1
P2M3_BlueGlueVacuum2	:INT:=197;	//3号叠台		备胶组件蓝胶真空2
P2M3_codeGlueVacuum1	:INT:=198;	//3号叠台		备胶组件二维码胶真空1
P2M3_codeGlueVacuum2	:INT:=199;	//3号叠台		备胶组件二维码胶真空2
P2M3_PastesGlueVacuum	:INT:=200;	//3号叠台		备胶组件贴胶头真空
P2M3_DTVacuum	:INT:=201;	//3号叠台		叠片台真空
P2M3_PoleSplintVacuum_D	:INT:=202;	//3号叠台		夹膜下夹板真空

P2M1_WJ_blow:INT:=203;//1号叠台 尾卷夹电芯吹气
P2M2_WJ_blow:INT:=204;//2号叠台 尾卷夹电芯吹气
P2M3_WJ_blow:INT:=205;//3号叠台 尾卷夹电芯吹气

P2M1_AnDTCarryingJRVacuum:INT:=206;//1号叠台 正极叠片搬运升降极耳真空
P2M2_AnDTCarryingJRVacuum:INT:=207;//2号叠台 正极叠片搬运升降极耳真空
P2M3_AnDTCarryingJRVacuum:INT:=208;//3号叠台 正极叠片搬运升降极耳真空

P2M1_CaDTCarryingJRVacuum:INT:=209;//1号叠台 负极叠片搬运升降极耳真空
P2M2_CaDTCarryingJRVacuum:INT:=210;//2号叠台 负极叠片搬运升降极耳真空
P2M3_CaDTCarryingJRVacuum:INT:=211;//3号叠台 负极叠片搬运升降极耳真空

P2M1_WJShortvacuum:INT:=212;//1短卷针张开真空
P2M2_WJShortvacuum:INT:=213;//2短卷针张开真空
P2M3_WJShortvacuum:INT:=214;//3短卷针张开真空
END_STRUCT
END_TYPE

// ---- P2DUTs/07_Name/ST_P2VirAxisName.TcDUT
TYPE ST_P2VirAxisName :   //虚轴名称
STRUCT
  
P2M1_VirTimeWind   	:INT:=140;	//P2M1时间虚轴
P2M1_VirMain	    :INT:=141;	//P2M1叠台主虚轴
P2M1_VirDriver	    :INT:=142;	//P2M1放卷驱动虚轴
P2M1_VirTailCurl	:INT:=143;	//P2M1尾卷虚轴
P2M1_VirGM	        :INT:=144;	//P2M1隔膜虚轴


P2M2_VirTimeWind   	:INT:=153;	//P2M2时间虚轴
P2M2_VirMain	:INT:=145;	//P2M2叠台主虚轴
P2M2_VirDriver	:INT:=146;	//P2M2放卷驱动虚轴
P2M2_VirTailCurl	:INT:=147;	//P2M2尾卷虚轴
P2M2_VirGM	        :INT:=148;	//P2M1隔膜虚轴			

P2M3_VirTimeWind   	:INT:=154;	//P2M3时间虚轴
P2M3_VirMain	:INT:=149;	//P2M3叠台主虚轴
P2M3_VirDriver	:INT:=150;	//P2M3放卷驱动虚轴
P2M3_VirTailCurl	:INT:=151;	//P2M3尾卷虚轴
P2M3_VirGM	        :INT:=152;	//P2M3隔膜虚轴			

END_STRUCT
END_TYPE

// ---- P2DUTs/07_Name/ST_RecName.TcDUT
TYPE ST_RecName :   //  整机纠偏名称
STRUCT
      P1PoleWind          :INT:=1; (***P1极片放卷纠偏*)
      P1PoleProcess      :INT:=2; (***P1极片放卷纠偏*)
      P1GMWind_U         :INT:=3; (***P1上隔膜纠偏*)
      P1GMWind_D         :INT:=4; (***P1下隔膜纠偏*)

      P2PoleWind_U          :INT:=5; (***P2上极片放卷纠偏*)
      P2PoleProcess_U      :INT:=6; (***P2上极片放卷纠偏*)
      P2PoleWind_D          :INT:=7; (***P2下极片放卷纠偏*)
      P2PoleProcess_D      :INT:=8; (***P2下极片放卷纠偏*)
      P2GMWind_U         :INT:=9; (***P2上隔膜纠偏*)
      P2GMWind_D         :INT:=10; (***P2下隔膜纠偏*)

      P3PoleWind_U          :INT:=11; (***P2上极片放卷纠偏*)
      P3PoleProcess_U      :INT:=12; (***P2上极片放卷纠偏*)
      P3PoleWind_D          :INT:=13; (***P2下极片放卷纠偏*)
      P3PoleProcess_D      :INT:=14; (***P2下极片放卷纠偏*)



END_STRUCT
END_TYPE

// ---- P2DUTs/07_Name/ST_TableName.TcDUT
TYPE ST_TableName :           //凸轮表
STRUCT
 	  M1_GMDanserMove_L	              :UINT:=100;	//1号叠台	隔膜摆臂左凸轮
	  M1_GMDanserMove_R	              :UINT:=101;	//1号叠台	隔膜摆臂左凸轮
      M1_GMWind_L	                          :UINT:=102;	//1号叠台	隔膜放卷左凸轮
      M1_GMWind_R	                      :UINT:=103;	//1号叠台	隔膜放卷右凸轮
  	  M1_GMBuffer_L	                      :UINT:=104;	//1号叠台	隔膜缓存左凸轮
      M1_GMBuffer_R	                      :UINT:=105;	//1号叠台	隔膜缓存右凸轮
  	  M1_GMLengthCalculate_L	           :UINT:=106;	//1号叠台	隔膜长度计算左凸轮
      M1_GMLengthCalculate_R	           :UINT:=107;	//1号叠台	隔膜长度计算右凸轮
      M1_AnCarryingLine                   	              :UINT:=108;	//1号叠台	正极送片搬运平移
	  
      M1_AnCarryingUpDown            	              :UINT:=109;	//1号叠台	正极送片搬运升降取片
      M1_AnCarryingUpDown1            	              :UINT:=110;	//1号叠台	正极送片搬运升降放片
	  M1_AnCarryingUpDown3            	              :UINT:=231;	//1号叠台	正极送片搬运升降放片    0240528SJ
      M1_AnCarryingWhirling             	              :UINT:=111;	//1号叠台	正极送片搬运旋转
      M1_AnDTCarryingLine                 	              :UINT:=112;	//1号叠台	正极叠台搬运平移1
      M1_AnDTCarryingUpDown           	              :UINT:=113;	//1号叠台	正极叠台搬运升降取片
      M1_AnDTCarryingUpDown1           	              :UINT:=114;	//1号叠台	正极叠台搬运升降放片
	  M1_AnDTCarryingUpDown3           	              :UINT:=232;	//1号叠台	正极叠台搬运升降放片    20240528SJ
      M1_CaCarryingLine1                    	              :UINT:=115;	//1号叠台	负极送片搬运1平移
      M1_CaCarryingUpDown1           	              :UINT:=116;	//1号叠台	负极送片搬运1升降
      M1_CaCarryingWhirling1           	              :UINT:=117;	//1号叠台	负极送片搬运1旋转
      M1_CaCarryingLine2                   	              :UINT:=118;	//1号叠台	负极送片搬运2平移
      M1_CaCarryingUpDown2             	              :UINT:=119;	//1号叠台	负极送片搬运2升降取片
      M1_CaCarryingUpDown2_1            	              :UINT:=120;	//1号叠台	负极送片搬运2升降放片
	   M1_CaCarryingUpDown2_3            	              :UINT:=233;	//1号叠台	负极送片搬运2升降放片  20240528SJ
      M1_CaBelt                                 	              :UINT:=121;	//1号叠台	负极送片皮带
      M1_CaDTCarryingLine                 	              :UINT:=122;	//1号叠台	负极叠台搬运平移
      M1_CaDTCarryingUpDown           	              :UINT:=123;	//1号叠台	负极叠台搬运升降取片
      M1_CaDTCarryingUpDown1          	              :UINT:=124;	//1号叠台	负极叠台搬运升降放片
	   M1_CaDTCarryingUpDown3          	              :UINT:=234;	//1号叠台	负极叠台搬运升降放片  20240528SJ
      M1_DTUpDown	              :UINT:=125;	//1号叠台	叠台升降
      M1_LeftYDLine                          	              :UINT:=126;	//1号叠台	左压刀开合
      M1_LeftYDUpDown                    	              :UINT:=127;	//1号叠台	左压刀升降
      M1_RightYDLine	              :UINT:=128;	//1号叠台	右压刀开合
      M1_RightYDUpDown                  	              :UINT:=129;	//1号叠台	右压刀升降
      M1_TailCurlLine                        	              :UINT:=130;	//1号叠台	尾卷平移
      M1_TailCurlUpDown	              :UINT:=131;	//1号叠台	尾卷升降
      M1_GMVir_L                            :UINT:=132;	//1号叠台  隔膜虚轴
 
	  M1_GMWind2_R                                     :UINT:=133;	
      M1_GMWind2_L                                      :UINT:=134;	
      M1_GMBuffer2_R                                   :UINT:=135;	
       M1_GMBuffer2_L                                    :UINT:=136;	
      M1_GMLengthCalculate2_R                      :UINT:=137;	
      M1_GMLengthCalculate2_L                      :UINT:=138;	
	  
	  
	  
	  
	  
  	  M2_GMDanserMove_L	              :UINT:=140;	//2号叠台	隔膜摆臂左凸轮
      M2_GMDanserMove_R	              :UINT:=141;	//2号叠台	隔膜摆臂左凸轮
      M2_GMWind_L	              :UINT:=142;	//2号叠台	隔膜放卷左凸轮
      M2_GMWind_R	              :UINT:=143;	//2号叠台	隔膜放卷右凸轮
      M2_GMBuffer_L	              :UINT:=144;	//2号叠台	隔膜缓存左凸轮
      M2_GMBuffer_R	              :UINT:=145;	//2号叠台	隔膜缓存右凸轮
      M2_GMLengthCalculate_L	              :UINT:=146;	//2号叠台	 隔膜长度计算左凸轮
      M2_GMLengthCalculate_R	              :UINT:=147;	//2号叠台	隔膜长度计算右凸轮
      M2_AnCarryingLine                  	              :UINT:=148;	//2号叠台	正极送片搬运平移
      M2_AnCarryingUpDown             	              :UINT:=149;	//2号叠台	正极送片搬运升降取片
      M2_AnCarryingUpDown1             	              :UINT:=150;	//2号叠台	正极送片搬运升降放片
	  M2_AnCarryingUpDown3             	              :UINT:=235;	//2号叠台	正极送片搬运升降放片  20240528SJ
      M2_AnCarryingWhirling              	              :UINT:=151;	//2号叠台	正极送片搬运旋转
      M2_AnDTCarryingLine               	              :UINT:=152;	//2号叠台	正极叠台搬运平移1
      M2_AnDTCarryingUpDown          	              :UINT:=153;	//2号叠台	正极叠台搬运升降取片
      M2_AnDTCarryingUpDown1           	              :UINT:=154;	//2号叠台	正极叠台搬运升降放片
	     M2_AnDTCarryingUpDown3           	          :UINT:=236;	//2号叠台	正极叠台搬运升降放片  20240528SJ
      M2_CaCarryingLine1                    	              :UINT:=155;	//2号叠台	负极送片搬运1平移
      M2_CaCarryingUpDown1              	              :UINT:=156;	//2号叠台	负极送片搬运1升降
      M2_CaCarryingWhirling1            	              :UINT:=157;	//2号叠台	负极送片搬运1旋转
      M2_CaCarryingLine2                   	              :UINT:=158;	//2号叠台	负极送片搬运2平移
      M2_CaCarryingUpDown2            	              :UINT:=159;	//2号叠台	负极送片搬运2升降取片
      M2_CaCarryingUpDown2_1             	              :UINT:=160;	//2号叠台	负极送片搬运2升降放片
	     M2_CaCarryingUpDown2_3             	              :UINT:=237;	//2号叠台	负极送片搬运2升降放片  20240528SJ
      M2_CaBelt                                  	              :UINT:=161;	//2号叠台	负极送片皮带
      M2_CaDTCarryingLine              	              :UINT:=162;	//2号叠台	负极叠台搬运平移
      M2_CaDTCarryingUpDown        	              :UINT:=163;	//2号叠台	负极叠台搬运升降取片
      M2_CaDTCarryingUpDown1         	              :UINT:=164;	//2号叠台	负极叠台搬运升降放片
	  M2_CaDTCarryingUpDown3         	              :UINT:=238;	//2号叠台	负极叠台搬运升降放片   20240528SJ
      M2_DTUpDown	              :UINT:=165;	//2号叠台	叠台升降
      M2_LeftYDLine                           	              :UINT:=166;	//2号叠台	左压刀开合
      M2_LeftYDUpDown                   	              :UINT:=167;	//2号叠台	左压刀升降
      M2_RightYDLine	              :UINT:=168;	//2号叠台	右压刀开合
      M2_RightYDUpDown                  	              :UINT:=169;	//2号叠台	右压刀升降
      M2_TailCurlLine                        	              :UINT:=170;	//2号叠台	尾卷平移
      M2_TailCurlUpDown	              :UINT:=171;	//2号叠台	尾卷升降
      M2_GMVir_L                            :UINT:=172;	//1号叠台  隔膜虚轴
 
 	  M2_GMWind2_R                                     :UINT:=173;	
	  M2_GMWind2_L                                      :UINT:=174;	
	  M2_GMBuffer2_R                                   :UINT:=175;	
	  M2_GMBuffer2_L                                    :UINT:=176;	
	  M2_GMLengthCalculate2_R                      :UINT:=177;	
	  M2_GMLengthCalculate2_L                      :UINT:=178;		
	  	  
	  
      M3_GMDanserMove_L	              :UINT:=180;	// 3号叠台 	隔膜摆臂左凸轮
      M3_GMDanserMove_R	              :UINT:=181;	// 3号叠台 	隔膜摆臂左凸轮
      M3_GMWind_L	              :UINT:=182;	// 3号叠台	隔膜放卷左凸轮
      M3_GMWind_R	              :UINT:=183;	// 3号叠台	隔膜放卷右凸轮
      M3_GMBuffer_L	              :UINT:=184;	// 3号叠台	隔膜缓存左凸轮
      M3_GMBuffer_R	              :UINT:=185;	// 3号叠台	隔膜缓存右凸轮
      M3_GMLengthCalculate_L	              :UINT:=186;	// 3号叠台	隔膜长度计算左凸轮
      M3_GMLengthCalculate_R	              :UINT:=187;	// 3号叠台	隔膜长度计算右凸轮
      M3_AnCarryingLine                   	              :UINT:=188;	// 3号叠台	正极送片搬运平移
      M3_AnCarryingUpDown          	              :UINT:=189;	// 3号叠台	正极送片搬运升降取片
      M3_AnCarryingUpDown1             	              :UINT:=190;	// 3号叠台	正极送片搬运升降放片
	  M3_AnCarryingUpDown3             	              :UINT:=239;	// 3号叠台	正极送片搬运升降放片    20240528SJ
      M3_AnCarryingWhirling             	              :UINT:=191;	// 3号叠台	正极送片搬运旋转
      M3_AnDTCarryingLine               	              :UINT:=192;	// 3号叠台	正极叠台搬运平移1
      M3_AnDTCarryingUpDown           	              :UINT:=193;	// 3号叠台	正极叠台搬运升降取片
      M3_AnDTCarryingUpDown1           	              :UINT:=194;	// 3号叠台	正极叠台搬运升降放片
	  M3_AnDTCarryingUpDown3           	              :UINT:=240;	// 3号叠台	正极叠台搬运升降放片 20240528SJ
      M3_CaCarryingLine1                   	              :UINT:=195;	// 3号叠台	负极送片搬运1平移
      M3_CaCarryingUpDown1              	              :UINT:=196;	// 3号叠台	负极送片搬运1升降
      M3_CaCarryingWhirling1            	              :UINT:=197;	// 3号叠台	负极送片搬运1旋转
      M3_CaCarryingLine2                    	              :UINT:=198;	// 3号叠台	负极送片搬运2平移
      M3_CaCarryingUpDown2            	              :UINT:=199;	// 3号叠台	负极送片搬运2升降取片
      M3_CaCarryingUpDown2_1             	              :UINT:=200;	// 3号叠台	负极送片搬运2升降放片
	  M3_CaCarryingUpDown2_3             	              :UINT:=241;	// 3号叠台	负极送片搬运2升降放片  20240528SJ  
      M3_CaBelt                                   	              :UINT:=201;	// 3号叠台	负极送片皮带
      M3_CaDTCarryingLine                  	              :UINT:=202;	// 3号叠台	负极叠台搬运平移
      M3_CaDTCarryingUpDown           	              :UINT:=203;	// 3号叠台	负极叠台搬运升降取片
      M3_CaDTCarryingUpDown1           	              :UINT:=204;	// 3号叠台	负极叠台搬运升降放片
	   M3_CaDTCarryingUpDown3           	              :UINT:=242;	// 3号叠台	负极叠台搬运升降放片   20240528SJ  
      M3_DTUpDown	              :UINT:=205;	// 3号叠台	叠台升降
      M3_LeftYDLine                             	              :UINT:=206;	// 3号叠台	左压刀开合
      M3_LeftYDUpDown                     	              :UINT:=207;	// 3号叠台	左压刀升降
      M3_RightYDLine	              :UINT:=208;	// 3号叠台	右压刀开合
      M3_RightYDUpDown                     	              :UINT:=209;	// 3号叠台	右压刀升降
	  M3_TailCurlLine                        	              :UINT:=210;	// 3号叠台	尾卷平移
 	  M3_TailCurlUpDown	              :UINT:=211;	// 3号叠台	尾卷升降
      M3_GMVir_L                            :UINT:=212;	//3号叠台  隔膜虚轴

	  
	  	M3_GMWind2_R                                     :UINT:=213;	
		M3_GMWind2_L                                      :UINT:=214;	
		M3_GMBuffer2_R                                   :UINT:=215;	
		M3_GMBuffer2_L                                    :UINT:=216;	
		M3_GMLengthCalculate2_R                      :UINT:=217;	
		M3_GMLengthCalculate2_L                      :UINT:=218;		

	  M1_LeftYDLine2                             	   :UINT:=219;	// 1号叠台	左压刀开合2
      M1_LeftYDUpDown2                     	           :UINT:=220;	// 1号叠台	左压刀升降2
      M1_RightYDLine2	                               :UINT:=221;	// 1号叠台	右压刀开合2
      M1_RightYDUpDown2                    	           :UINT:=222;	// 1号叠台	右压刀升降2
	  
	  M2_LeftYDLine2                             	   :UINT:=223;	// 2号叠台	左压刀开合2
      M2_LeftYDUpDown2                     	           :UINT:=224;	// 2号叠台	左压刀升降2
      M2_RightYDLine2	                               :UINT:=225;	// 2号叠台	右压刀开合2
      M2_RightYDUpDown2                    	           :UINT:=226;	// 2号叠台	右压刀升降2
	  
	  M3_LeftYDLine2                             	   :UINT:=227;	// 3号叠台	左压刀开合2
      M3_LeftYDUpDown2                     	           :UINT:=228;	// 3号叠台	左压刀升降2
      M3_RightYDLine2	                               :UINT:=229;	// 3号叠台	右压刀开合2
      M3_RightYDUpDown2                    	           :UINT:=230;	// 3号叠台	右压刀升降2	  
	  
	  
	  
	  
	  
	  
	  
END_STRUCT
END_TYPE

// ---- P2DUTs/07_Name/ST_VirAxisName.TcDUT
TYPE ST_VirAxisName :
STRUCT
	VirTimeWind	:INT;	//P2时间虚轴

	VirMain	:INT;	//叠台主虚轴
	VirDriver	:INT;	//放卷驱动虚轴

	VirTailCurl	:INT;	//尾卷虚轴

    VirGM  :INT ;  //隔膜虚轴

	CaCarryingVirGM  :INT ;  //负极取料虚轴


END_STRUCT
END_TYPE

// ---- P2DUTs/08_IO/ST_Button.TcDUT
TYPE ST_Button :
STRUCT
Tricolorlamp_Yellow 	:BOOL;		//		三色灯_黄
Tricolorlamp_Red 	:BOOL;		//		三色灯_绿
Tricolorlamp_Green 	:BOOL;		//		三色灯_红
Tricolorlamp_Buzzer	:BOOL;		//		三色灯_蜂鸣器
PoleInflationLights	:BOOL;		//		隔膜气胀轴按钮灯
PoleTapeSplicerLLights	:BOOL;		//		隔膜左压板气缸按钮灯
PoleTapeSplicerRLights	:BOOL;		//		隔膜右压板气缸按钮灯
BlueGlueLights	:BOOL;		//		压蓝胶按钮灯
codeGlueLights	:BOOL;		//		压二维码胶按钮灯
PoleInflationbtn	:BOOL;		//		隔膜气胀轴按钮
PoleTapeSplicerLbtn	:BOOL;		//		隔膜左压板气缸按钮
PoleTapeSplicerRbtn	:BOOL;		//		隔膜右压板气缸按钮
BlueGluebtn	:BOOL;		//		一键备蓝胶按钮
BlueGluebtnLights	:BOOL;		//		一键备蓝胶按钮灯
BlueGluePressbtn	:BOOL;		//		压蓝胶按钮
codeGluebtn	:BOOL;		//		一键备二维码胶按钮
codeGluebtnLights	:BOOL;		//		一键备二维码胶按钮灯
codeGluePressbtn	:BOOL;		//		压二维码胶按钮
EmStopbtn1	:BOOL;		//		外罩急停1
EmStopbtn2	:BOOL;		//		外罩急停2
EmStopbtn3	:BOOL;		//		外罩急停3
EmStopbtn4	:BOOL;		//		外罩急停4

END_STRUCT
END_TYPE

// ---- P2DUTs/08_IO/ST_P2Button.TcDUT
TYPE ST_P2Button ://P2 按钮
STRUCT
System_StartLights	:BOOL;	//		控制面板启动按钮灯
System_ResetLights	:BOOL;	//		控制面板复位按钮灯
System_StopLights	:BOOL;	//		控制面板停止按钮灯
System_Autonbtn	:BOOL;	//		控制面板手自动切换按钮
System_Startbtn	:BOOL;	//		控制面板启动按钮
System_Rrestbtn	:BOOL;	//		控制面板复位按钮
System_Stopbtn	:BOOL;	//		控制面板停止按钮
System_EmStopbtn	:BOOL;	//		控制面板急停按钮

P2M1_Tricolorlamp_Yellow 	:BOOL;	//1号叠台		三色灯_黄
P2M1_Tricolorlamp_Red 	:BOOL;	//1号叠台		三色灯_绿
P2M1_Tricolorlamp_Green 	:BOOL;	//1号叠台		三色灯_红
P2M1_Tricolorlamp_Buzzer	:BOOL;	//1号叠台		三色灯_蜂鸣器
P2M1_PoleInflationLights	:BOOL;	//1号叠台		隔膜气胀轴按钮灯
P2M1_PoleTapeSplicerLLights	:BOOL;	//1号叠台		隔膜左压板气缸按钮灯
P2M1_PoleTapeSplicerRLights	:BOOL;	//1号叠台		隔膜右压板气缸按钮灯
P2M1_BlueGlueLights	:BOOL;	//1号叠台		压蓝胶按钮灯
P2M1_codeGlueLights	:BOOL;	//1号叠台		压二维码胶按钮灯
P2M1_PoleInflationbtn	:BOOL;	//1号叠台		隔膜气胀轴按钮
P2M1_PoleTapeSplicerLbtn	:BOOL;	//1号叠台		隔膜左压板气缸按钮
P2M1_PoleTapeSplicerRbtn	:BOOL;	//1号叠台		隔膜右压板气缸按钮
P2M1_BlueGluebtn	:BOOL;	//1号叠台		一键备蓝胶按钮
P2M1_BlueGluebtnLights	:BOOL;	//1号叠台		一键备蓝胶按钮灯
P2M1_BlueGluePressbtn	:BOOL;	//1号叠台		压蓝胶按钮
P2M1_codeGluebtn	:BOOL;	//1号叠台		一键备二维码胶按钮
P2M1_codeGluebtnLights	:BOOL;	//1号叠台		一键备二维码胶按钮灯
P2M1_codeGluePressbtn	:BOOL;	//1号叠台		压二维码胶按钮
P2M1_EmStopbtn1	:BOOL;	//1号叠台		外罩急停1
P2M1_EmStopbtn2	:BOOL;	//1号叠台		外罩急停2
P2M1_EmStopbtn3	:BOOL;	//1号叠台		外罩急停3
P2M1_EmStopbtn4	:BOOL;	//1号叠台		外罩急停4
P2M1_Startbtn:BOOL;//1号叠台，启动按钮
P2M1_Resetebtn:BOOL;//1号叠台，复位按钮
P2M1_Stopbtn:BOOL;//1号叠台，停止按钮
P2M1_Autobtn:BOOL;//1号叠台，手自动按钮



P2M2_Tricolorlamp_Yellow 	:BOOL;	//2号叠台		三色灯_黄
P2M2_Tricolorlamp_Red 	:BOOL;	//2号叠台		三色灯_绿
P2M2_Tricolorlamp_Green 	:BOOL;	//2号叠台		三色灯_红
P2M2_Tricolorlamp_Buzzer	:BOOL;	//2号叠台		三色灯_蜂鸣器
P2M2_PoleInflationLights	:BOOL;	//2号叠台		隔膜气胀轴按钮灯
P2M2_PoleTapeSplicerLLights	:BOOL;	//2号叠台		隔膜左压板气缸按钮灯
P2M2_PoleTapeSplicerRLights	:BOOL;	//2号叠台		隔膜右压板气缸按钮灯
P2M2_BlueGlueLights	:BOOL;	//2号叠台		压蓝胶按钮灯
P2M2_codeGlueLights	:BOOL;	//2号叠台		压二维码胶按钮灯
P2M2_PoleInflationbtn	:BOOL;	//2号叠台		隔膜气胀轴按钮
P2M2_PoleTapeSplicerLbtn	:BOOL;	//2号叠台		隔膜左压板气缸按钮
P2M2_PoleTapeSplicerRbtn	:BOOL;	//2号叠台		隔膜右压板气缸按钮
P2M2_BlueGluebtnLights	:BOOL;	//2号叠台		一键备蓝胶按钮灯
P2M2_BlueGluebtn	:BOOL;	//2号叠台		一键备蓝胶按钮
P2M2_BlueGluePressbtn	:BOOL;	//2号叠台		压蓝胶按钮
P2M2_codeGluebtnLights	:BOOL;	//2号叠台		一键备二维码胶按钮灯
P2M2_codeGluebtn	:BOOL;	//2号叠台		一键备二维码胶按钮
P2M2_codeGluePressbtn	:BOOL;	//2号叠台		压二维码胶按钮
P2M2_EmStopbtn1	:BOOL;	//2号叠台		外罩急停1
P2M2_EmStopbtn2	:BOOL;	//2号叠台		外罩急停2
P2M2_EmStopbtn3	:BOOL;	//2号叠台		外罩急停3
P2M2_EmStopbtn4	:BOOL;	//2号叠台		外罩急停4
P2M2_Startbtn:BOOL;//2号叠台，启动按钮
P2M2_Resetebtn:BOOL;//2号叠台，复位按钮
P2M2_Stopbtn:BOOL;//2号叠台，停止按钮
P2M2_Autobtn:BOOL;//2号叠台，手自动按钮


P2M3_Tricolorlamp_Yellow 	:BOOL;	//2号叠台		三色灯_黄
P2M3_Tricolorlamp_Red 	:BOOL;	//2号叠台		三色灯_绿
P2M3_Tricolorlamp_Green 	:BOOL;	//2号叠台		三色灯_红
P2M3_Tricolorlamp_Buzzer	:BOOL;	//2号叠台		三色灯_蜂鸣器
P2M3_PoleInflationLights	:BOOL;	//3号叠台		隔膜气胀轴按钮灯
P2M3_PoleTapeSplicerLLights	:BOOL;	//3号叠台		隔膜左压板气缸按钮灯
P2M3_PoleTapeSplicerRLights	:BOOL;	//3号叠台		隔膜右压板气缸按钮灯
P2M3_BlueGlueLights	:BOOL;	//3号叠台		压蓝胶按钮灯
P2M3_codeGlueLights	:BOOL;	//3号叠台		压二维码胶按钮灯
P2M3_PoleInflationbtn	:BOOL;	//3号叠台		隔膜气胀轴按钮
P2M3_PoleTapeSplicerLbtn	:BOOL;	//3号叠台		隔膜左压板气缸按钮
P2M3_PoleTapeSplicerRbtn	:BOOL;	//3号叠台		隔膜右压板气缸按钮
P2M3_BlueGluebtnLights	:BOOL;	//3号叠台		一键备蓝胶按钮灯
P2M3_BlueGluebtn	:BOOL;	//3号叠台		一键备蓝胶按钮
P2M3_BlueGluePressbtn	:BOOL;	//3号叠台		压蓝胶按钮
P2M3_codeGluebtnLights	:BOOL;	//3号叠台		一键备二维码胶按钮灯
P2M3_codeGluebtn	:BOOL;	//3号叠台		一键备二维码胶按钮
P2M3_codeGluePressbtn	:BOOL;	//3号叠台		压二维码胶按钮
P2M3_EmStopbtn1	:BOOL;	//3号叠台		外罩急停1
P2M3_EmStopbtn2	:BOOL;	//3号叠台		外罩急停2
P2M3_EmStopbtn3	:BOOL;	//3号叠台		外罩急停3
P2M3_EmStopbtn4	:BOOL;	//3号叠台		外罩急停4
P2M3_Startbtn:BOOL;//3号叠台，启动按钮
P2M3_Resetebtn:BOOL;//3号叠台，复位按钮
P2M3_Stopbtn:BOOL;//3号叠台，停止按钮
P2M3_Autobtn:BOOL;//3号叠台，手自动按钮


P2M3_Securitydoorswitch8	:BOOL;	//3号叠台		外罩门禁8
END_STRUCT
END_TYPE

// ---- P2DUTs/08_IO/ST_P2Senser.TcDUT
TYPE ST_P2Senser ://P2 传感器
STRUCT
NGBatteries_H:BOOL;//电芯NG1料盒高度感应
NGBatteries_L:BOOL;//电芯NG1料盒到位感应
P2M1_AnBeltsensor	:BOOL;	//1号叠台		正极模切送料分段皮带1有料感应
P2M1_CaBeltsensor	:BOOL;	//1号叠台		负极模切送料分段皮带1有料感应
P2M1_Offloadingsensor	:BOOL;	//1号叠台		取料位感应
P2M1_BlueGluetsensor	:BOOL;	//1号叠台		蓝胶料盘检测
P2M1_codeGluesensor	:BOOL;	//1号叠台		二维码胶料盘检测
P2M1_Markesensor	:BOOL;	//1号叠台		二维码胶Mark孔检测
P2M1_GluebHave      :BOOL;  //1号叠台		一号贴胶旋转电芯感应
P2M1_Coldpressingesensor	:BOOL;	//1号叠台		冷压上料夹平移电机1号叠台处检测
P2M1_Securitydoorswitch1	:BOOL;	//1号叠台		外罩门禁1
P2M1_Securitydoorswitch2	:BOOL;	//1号叠台		外罩门禁2
P2M1_Securitydoorswitch3	:BOOL;	//1号叠台		外罩门禁3
P2M1_Securitydoorswitch4	:BOOL;	//1号叠台		外罩门禁4
P2M1_Securitydoorswitch5	:BOOL;	//1号叠台		外罩门禁5
P2M1_Securitydoorswitch6	:BOOL;	//1号叠台		外罩门禁6
P2M1_Securitydoorswitch7	:BOOL;	//1号叠台		外罩门禁7
P2M1_Securitydoorswitch8	:BOOL;	//1号叠台		外罩门禁8
P2M1_Securitydoorswitch9	:BOOL;	//1号叠台		外罩门禁9
P2M1_Securitydoorswitch10	:BOOL;	//1号叠台		外罩门禁10
P2M1_Yellowmark       :BOOL;  //1号叠台		一号隔膜黄标感应    
P2M1_Ceramics:BOOL;// //1号叠台		一号隔膜陶瓷面检测    
P2M1_AnDTCarryingJROnSwitch:BOOL;//1号正极极耳真空信号
P2M1_CaDTCarryingJROnSwitch:BOOL;//1号负极极耳真空信号
P2M1_AnNGboxsensor 	:BOOL;		//1叠台正极NG料盒满料感应
P2M1_CaNGboxsensor 	:BOOL;		//1叠台负极NG料盒满料感应

P2M2_AnBeltsensor	:BOOL;	//2号叠台		正极模切送料分段皮带1有料感应
P2M2_CaBeltsensor	:BOOL;	//2号叠台		负极模切送料分段皮带1有料感应
P2M2_Offloadingsensor	:BOOL;	//2号叠台		取料位感应
P2M2_BlueGluetsensor	:BOOL;	//2号叠台		蓝胶料盘检测
P2M2_codeGluesensor	:BOOL;	//2号叠台		二维码胶料盘检测
P2M2_Markesensor	:BOOL;	//2号叠台		二维码胶Mark孔检测
P2M2_GluebHave      :BOOL;  //2号叠台		二号贴胶旋转电芯感应
P2M2_Coldpressingesensor	:BOOL;	//2号叠台		冷压上料夹平移电机1号叠台处检测
P2M2_Securitydoorswitch1	:BOOL;	//2号叠台		外罩门禁1
P2M2_Securitydoorswitch2	:BOOL;	//2号叠台		外罩门禁2
P2M2_Securitydoorswitch3	:BOOL;	//2号叠台		外罩门禁3
P2M2_Securitydoorswitch4	:BOOL;	//2号叠台		外罩门禁4
P2M2_Securitydoorswitch5	:BOOL;	//2号叠台		外罩门禁5
P2M2_Securitydoorswitch6	:BOOL;	//2号叠台		外罩门禁6
P2M2_Securitydoorswitch7	:BOOL;	//2号叠台		外罩门禁7
P2M2_Securitydoorswitch8	:BOOL;	//2号叠台		外罩门禁8
P2M2_Securitydoorswitch9	:BOOL;	//2号叠台		外罩门禁9
P2M2_Securitydoorswitch10	:BOOL;	//2号叠台		外罩门禁10
P2M2_Yellowmark       :BOOL;  //2号叠台		二号隔膜黄标感应    
P2M2_Ceramics:BOOL;// //1号叠台		2号隔膜陶瓷面检测   
P2M2_AnDTCarryingJROnSwitch:BOOL;//2号正极极耳真空信号
P2M2_CaDTCarryingJROnSwitch:BOOL;//2号负极极耳真空信号 
P2M2_AnNGboxsensor 	:BOOL;		//2叠台正极NG料盒满料感应
P2M2_CaNGboxsensor 	:BOOL;		//2叠台负极NG料盒满料感应

P2M3_AnBeltsensor	:BOOL;	//3号叠台		正极模切送料分段皮带1有料感应
P2M3_CaBeltsensor	:BOOL;	//3号叠台		负极模切送料分段皮带1有料感应
P2M3_Offloadingsensor	:BOOL;	//3号叠台		取料位感应
P2M3_BlueGluetsensor	:BOOL;	//3号叠台		蓝胶料盘检测
P2M3_codeGluesensor	:BOOL;	//3号叠台		二维码胶料盘检测
P2M3_Markesensor	:BOOL;	//3号叠台		二维码胶Mark孔检测
P2M3_GluebHave      :BOOL;  //3号叠台	    三号贴胶旋转电芯感应
P2M3_Coldpressingesensor	:BOOL;	//3号叠台		冷压上料夹平移电机1号叠台处检测
P2M3_Securitydoorswitch1	:BOOL;	//3号叠台		外罩门禁1
P2M3_Securitydoorswitch2	:BOOL;	//3号叠台		外罩门禁2
P2M3_Securitydoorswitch3	:BOOL;	//3号叠台		外罩门禁3
P2M3_Securitydoorswitch4	:BOOL;	//3号叠台		外罩门禁4
P2M3_Securitydoorswitch5	:BOOL;	//3号叠台		外罩门禁5
P2M3_Securitydoorswitch6	:BOOL;	//3号叠台		外罩门禁6
P2M3_Securitydoorswitch7	:BOOL;	//3号叠台		外罩门禁7
P2M3_Securitydoorswitch8	:BOOL;	//3号叠台		外罩门禁8
P2M3_Securitydoorswitch9	:BOOL;	//3号叠台		外罩门禁9
P2M3_Securitydoorswitch10	:BOOL;	//3号叠台		外罩门禁10



P2M3_Yellowmark       :BOOL;  //3号叠台		三号隔膜黄标感应    
P2M3_Ceramics:BOOL;// //3号叠台		3号隔膜陶瓷面检测    
P2M3_AnDTCarryingJROnSwitch:BOOL;//3号正极极耳真空信号
P2M3_CaDTCarryingJROnSwitch:BOOL;//3号负极极耳真空信号
P2M3_AnNGboxsensor 	:BOOL;		//3叠台正极NG料盒满料感应
P2M3_CaNGboxsensor 	:BOOL;		//3叠台负极NG料盒满料感应
END_STRUCT
END_TYPE

// ---- P2DUTs/08_IO/ST_Senser.TcDUT
TYPE ST_Senser :
STRUCT
AnBeltsensor	:BOOL;		//		正极模切送料分段皮带1有料感应
AnLimitSwitch:BOOL;//正极取片搬运、叠片搬运防撞感应
CaBeltsensor	:BOOL;		//		负极模切送料分段皮带1有料感应
CaLimitSwitch:BOOL;//负极取片搬运、叠片搬运防撞感应
Offloadingsensor	:BOOL;		//		取料位感应
BlueGluetsensor	:BOOL;		//		蓝胶料盘检测
codeGluesensor	:BOOL;		//		二维码胶料盘检测
Markesensor	:BOOL;		//		二维码胶Mark孔检测
GluebHave	:BOOL;		//		贴胶旋转电芯感应
Coldpressingesensor		:BOOL;		//		冷压上料夹平移电机1号叠台处检测
Securitydoorswitch1		:BOOL;		//		外罩门禁1
Securitydoorswitch2		:BOOL;		//		外罩门禁2
Securitydoorswitch3		:BOOL;		//		外罩门禁3
Securitydoorswitch4		:BOOL;		//		外罩门禁4
Securitydoorswitch5		:BOOL;		//		外罩门禁5
Securitydoorswitch6		:BOOL;		//		外罩门禁6
Securitydoorswitch7		:BOOL;		//		外罩门禁7
Securitydoorswitch8		:BOOL;		//		外罩门禁8
Securitydoorswitch9		:BOOL;		//		外罩门禁9
Securitydoorswitch10	:BOOL;		//		外罩门禁10
QYcode  :BOOL;//叠台储气罐真空信号
Yellowmark       :BOOL;  //叠台隔膜黄标感应    
Ceramics:BOOL;//隔膜陶瓷面感应器
AnDTCarryingJROnSwitch:BOOL;//正极极耳真空信号
CaDTCarryingJROnSwitch:BOOL;//负极极耳真空信号
AnNGboxsensor 	:BOOL;		//叠台正极NG料盒满料感应
CaNGboxsensor 	:BOOL;		//叠台负极NG料盒满料感应

END_STRUCT
END_TYPE

// ---- P2DUTs/08_IO/ST_SystemButton.TcDUT
TYPE ST_SystemButton :
STRUCT
System_StartLights	:BOOL;		//		控制面板启动按钮灯
System_ResetLights	:BOOL;		//		控制面板复位按钮灯
System_StopLights	:BOOL;		//		控制面板停止按钮灯
System_Autonbtn	:BOOL;		//		控制面板手自动切换按钮
System_Startbtn	:BOOL;		//		控制面板启动按钮
System_Rrestbtn	:BOOL;		//		控制面板复位按钮
System_Stopbtn	:BOOL;		//		控制面板停止按钮
System_EmStopbtn	:BOOL;		//		控制面板急停按钮

END_STRUCT
END_TYPE

// ---- P2DUTs/08_IO/System_Senser.TcDUT
TYPE System_Senser :
STRUCT
END_STRUCT
END_TYPE

// ---- P2DUTs/30_Parameter/04_Rectify/ST_PLC_PC_MES.TcDUT
TYPE ST_PLC_PC_MES  :
STRUCT
//PC写给PLC的-----先下发给叠台，叠台再和模切做通讯-------需要上料时PLC往该地址写入Error
PostiveCode1				:STRING(49);//正极左1条码		1
PostiveCode2				:STRING(49);//正极右2条码		2
NegativeCode1				:STRING(49);//负极左1条码		3
NegativeCode2				:STRING(49);//负极右2条码		4
Station1_Code				:STRING(49);//叠台1隔膜条码		5
Station2_Code				:STRING(49);//叠台2隔膜条码		6
Station3_Code				:STRING(49);//叠台3隔膜条码		7
Station1_BlueCode			:STRING(49);//叠台1l蓝胶条码		8
Station2_BlueCode			:STRING(49);//叠台2蓝胶条码		9
Station3_BlueCode			:STRING(49);//叠台3蓝胶条码		10
CellCode					:STRING(49);//后段二维码胶条码	11
BlueCode					:STRING(49);//后段蓝胶条码		12

//MES条码校验信号交互----PC_To_PLC
Mes_PcToPlc1:        BOOL;   //正极左1条码条码校验完成信号
Mes_PcToPlc2:        BOOL;   //正极右2条码校验完成信号
Mes_PcToPlc3:        BOOL;   //负极左1条码	校验完成信号
Mes_PcToPlc4:        BOOL;   //负极右2条码校验完成信号
Mes_PcToPlc5:        BOOL;   //叠台1隔膜条码校验完成信号
Mes_PcToPlc6:        BOOL;   //叠台2隔膜条码校验完成信号
Mes_PcToPlc7:        BOOL;   //叠台3隔膜条码校验完成信号
Mes_PcToPlc8:        BOOL;   //叠台1l蓝胶条码校验完成信号
Mes_PcToPlc9:        BOOL;   //叠台2蓝胶条码校验完成信号
Mes_PcToPlc10:        BOOL;  //叠台3蓝胶条码校验完成信号
Mes_PcToPlc11:        BOOL;   //后段二维码胶条码校验完成信号
Mes_PcToPlc12:        BOOL;   //后段蓝胶条码校验完成信号	

END_STRUCT
END_TYPE

// ---- P2DUTs/30_Parameter/04_Rectify/ST_RecCmd.TcDUT
TYPE ST_RecCmd ://过程纠偏
STRUCT
    bLock:				BOOL;	//纠偏外部锁定
	bAuto:				BOOL;	//纠偏自动
	bManual:           BOOL;  //纠偏手动
	bCentre:           BOOL;	//纠偏居中

END_STRUCT
END_TYPE

// ---- P2DUTs/30_Parameter/04_Rectify/ST_RecCtrl.TcDUT
TYPE ST_RecCtrl ://过程纠偏
STRUCT
    Cmd        :ST_RecCmd;
    Io            :ST_RecIo;
    Status      :ST_RecStatus;
END_STRUCT
END_TYPE

// ---- P2DUTs/30_Parameter/04_Rectify/ST_RecIo.TcDUT
TYPE ST_RecIo ://过程纠偏
STRUCT
	biError:				BOOL;	//纠偏报警
	biCentre:           BOOL;	//纠偏居中状态  

	
    boLock:				BOOL;	//纠偏外部锁定
	boAuto:				BOOL;	//纠偏自动
	boManual:           BOOL;  //纠偏手动
	boCentre:           BOOL;	//纠偏居中

END_STRUCT
END_TYPE

// ---- P2DUTs/30_Parameter/04_Rectify/ST_RecStatus.TcDUT
TYPE ST_RecStatus ://过程纠偏
STRUCT
    bError             :BOOL;     //纠偏故障
    bRuning           :BOOL;    //纠偏运行中
END_STRUCT
END_TYPE

// ---- P2DUTs/30_Parameter/ST_DT_To_MQ_MES.TcDUT
TYPE ST_DT_To_MQ_MES  :
STRUCT
//PC写给PLC的-----先下发给叠台，叠台再和模切做通讯-------需要上料时PLC往该地址写入Error
PostiveCode1				:STRING(49);//正极左1条码		1
PostiveCode2				:STRING(49);//正极右2条码		2
NegativeCode1				:STRING(49);//负极左1条码		3
NegativeCode2				:STRING(49);//负极右2条码		4
Station1_Code				:STRING(49);//叠台1隔膜条码		5
Station2_Code				:STRING(49);//叠台2隔膜条码		6
Station3_Code				:STRING(49);//叠台3隔膜条码		7
Station1_BlueCode			:STRING(49);//叠台1l蓝胶条码		8
Station2_BlueCode			:STRING(49);//叠台2蓝胶条码		9
Station3_BlueCode			:STRING(49);//叠台3蓝胶条码		10
CellCode					:STRING(49);//后段二维码胶条码	11
BlueCode					:STRING(49);//后段蓝胶条码		12

//MES条码校验信号交互----PC_To_PLC
Mes_PcToPlc1:        BOOL;   //正极左1条码条码校验完成信号
Mes_PcToPlc2:        BOOL;   //正极右2条码校验完成信号
Mes_PcToPlc3:        BOOL;   //负极左1条码	校验完成信号
Mes_PcToPlc4:        BOOL;   //负极右2条码校验完成信号
Mes_PcToPlc5:        BOOL;   //叠台1隔膜条码校验完成信号
Mes_PcToPlc6:        BOOL;   //叠台2隔膜条码校验完成信号
Mes_PcToPlc7:        BOOL;   //叠台3隔膜条码校验完成信号
Mes_PcToPlc8:        BOOL;   //叠台1l蓝胶条码校验完成信号
Mes_PcToPlc9:        BOOL;   //叠台2蓝胶条码校验完成信号
Mes_PcToPlc10:        BOOL;  //叠台3蓝胶条码校验完成信号
Mes_PcToPlc11:        BOOL;   //后段二维码胶条码校验完成信号
Mes_PcToPlc12:        BOOL;   //后段蓝胶条码校验完成信号	

//DT_To_MQ---清换卷触发信号
MesClear_Pc1:        BOOL;   //正极左1换料信号清理
MesClear_Pc2:        BOOL;   //正极右2换料信号清理
MesClear_Pc3:        BOOL;   //负极左1换料信号清理
MesClear_Pc4:        BOOL;   //负极右2换料信号清理

END_STRUCT
END_TYPE

// ---- P2DUTs/30_Parameter/ST_MQ_To_DT_MES.TcDUT
TYPE ST_MQ_To_DT_MES  :
STRUCT
//PC写给PLC的-----先下发给叠台，叠台再和模切做通讯-------需要上料时PLC往该地址写入Error
PostiveCode1				:STRING(49);//正极左1条码		1
PostiveCode2				:STRING(49);//正极右2条码		2
NegativeCode1				:STRING(49);//负极左1条码		3
NegativeCode2				:STRING(49);//负极右2条码		4
Station1_Code				:STRING(49);//叠台1隔膜条码		5
Station2_Code				:STRING(49);//叠台2隔膜条码		6
Station3_Code				:STRING(49);//叠台3隔膜条码		7
Station1_BlueCode			:STRING(49);//叠台1l蓝胶条码		8
Station2_BlueCode			:STRING(49);//叠台2蓝胶条码		9
Station3_BlueCode			:STRING(49);//叠台3蓝胶条码		10
CellCode					:STRING(49);//后段二维码胶条码	11
BlueCode					:STRING(49);//后段蓝胶条码		12

//MES条码校验信号交互----PC_To_PLC
Mes_PcToPlc1:        BOOL;   //正极左1条码条码校验完成信号
Mes_PcToPlc2:        BOOL;   //正极右2条码校验完成信号
Mes_PcToPlc3:        BOOL;   //负极左1条码	校验完成信号
Mes_PcToPlc4:        BOOL;   //负极右2条码校验完成信号
Mes_PcToPlc5:        BOOL;   //叠台1隔膜条码校验完成信号
Mes_PcToPlc6:        BOOL;   //叠台2隔膜条码校验完成信号
Mes_PcToPlc7:        BOOL;   //叠台3隔膜条码校验完成信号
Mes_PcToPlc8:        BOOL;   //叠台1l蓝胶条码校验完成信号
Mes_PcToPlc9:        BOOL;   //叠台2蓝胶条码校验完成信号
Mes_PcToPlc10:        BOOL;  //叠台3蓝胶条码校验完成信号
Mes_PcToPlc11:        BOOL;   //后段二维码胶条码校验完成信号
Mes_PcToPlc12:        BOOL;   //后段蓝胶条码校验完成信号	

//MES条码校验信号交互----PLC_To_PC
Mes_PlcToPc1:        BOOL;   //正极左1换料信号
Mes_PlcToPc2:        BOOL;   //正极右2换料信号
Mes_PlcToPc3:        BOOL;   //负极左1换料信号
Mes_PlcToPc4:        BOOL;   //负极右2换料信号
END_STRUCT
END_TYPE

// ---- P2DUTs/30_Parameter/ST_ParFilterAD.TcDUT
TYPE ST_ParFilterAD :  //P1部分参数
STRUCT
	iLimitH             :REAL;//转换前高限值
	iLimitL             :REAL;//转换前低限值
	fRangeH         :REAL;//量程高限
	fRangeL          :REAL;//量程低限
END_STRUCT
END_TYPE

// ---- P2DUTs/30_Parameter/ST_ParMachine.TcDUT
TYPE ST_ParMachine ://机械参数
STRUCT
(*
       fMQDriverDiameter            :REAL:=80   ;
      
       fYFHDriverInDiameter         :REAL:=24   ;  //预复合入料辊直径
       fAuxDriverDiameter            :REAL:=64 ;  //辅助驱动辊张力

       fYFHGMDriverDiameter      :REAL:=64 ; //预复合隔膜压辊直径
       fYFHGMDriverDiameter2      :REAL:=32 ; 



       fMainRollDriverDiameter       :REAL:=200 ;//复合大辊直径

      fP4MainDriverDiameter        :REAL:=70 ;//P4主驱动
      fP4AuxDriverDiameter        :REAL:=30 ;//P4f辅驱动




//叠片主驱动  70
//叠片辅驱动  30
//NG皮带 46




















*)









END_STRUCT
END_TYPE

// ---- P2DUTs/30_Parameter/ST_ParProduct.TcDUT
TYPE ST_ParProduct ://工艺参数
STRUCT
(*
         fAnPoleWith                            :REAL:=98 ;    //正极片宽
         fCaPoleWith                            :REAL:=100;   //负极片宽
         fGMInterval                            :REAL:=2 ;     //隔膜间距
         iRunMode                               :UINT;   //运行模式    1：空跑隔膜    2：不带隔膜整机空跑   3：只跑1#      4::连续制片模式     5：标准模式      
         iMainVel                                  :UINT;  //运行速度 PPM (最大值180)          整机效率=iMainVel*4  

         
       

        Publ:                                       	ST_ParPublic;   
        P2M1:                                          ST_P2Par; (******P2 部分参数******)
		P2M2:                                          ST_P2Par; (******P2 部分参数******)
		P2M3:                                          ST_P2Par; (******P2 部分参数******)
*)
END_STRUCT
END_TYPE

// ---- P2DUTs/30_Parameter/ST_ParTableNo.TcDUT
TYPE ST_ParTableNo ://    凸轮表号
STRUCT
(*
P2M1AnCarryingLine1     	 	 :UINT :=10;	//1号叠台	正极搬运平移凸轮号从取料位到叠台位
P2M1AnCarryingLine2   		 :UINT :=11;	//1号叠台	正极搬运平移凸轮号从叠台位到取料位
P2M1AnDTCarryingLine1		 :UINT :=12;	//1号叠台	正极叠台搬运平移凸轮从取料位到叠台位
P2M1AnDTCarryingLine2		 :UINT :=13;	//1号叠台	正极叠台搬运平移凸轮从叠台位到取料位
P2M1AnCarryingUpdown1		 :UINT :=14;	//1号叠台	正极搬运升降凸轮从取料位到叠台位
P2M1AnCarryingUpdown2		 :UINT :=15;	//1号叠台	正极搬运升降凸轮从叠台位到取料位
P2M1AnDTCarryingUpDown1		 :UINT :=16;	//1号叠台	正极叠台搬运升降凸轮从取料位到叠台位
P2M1AnDTCarryingUpDown2		 :UINT :=17;	//1号叠台	正极叠台搬运升降凸轮从叠台位到取料位
P2M1AnCarryingWhirling1		 :UINT :=18;	//1号叠台	正极搬运旋转凸轮从取料位到叠台位
P2M1AnCarryingWhirling2		 :UINT :=19;	//1号叠台	正极搬运旋转凸轮从叠台位到取片位
P2M1CaCarryingLine1     	 	 :UINT :=20;	//1号叠台	负极搬运平移凸轮号从取料位到叠台位
P2M1CaCarryingLine2   		 :UINT :=21;	//1号叠台	负极搬运平移凸轮号从叠台位到取料位
P2M1CaDTCarryingLine1		 :UINT :=22;	//1号叠台	负极叠台搬运平移凸轮从取料位到叠台位
P2M1CaDTCarryingLine2		 :UINT :=23;	//1号叠台	负极叠台搬运平移凸轮从叠台位到取料位
P2M1CaCarryingUpdown1		 :UINT :=24;	//1号叠台	负极搬运升降凸轮从取料位到叠台位
P2M1CaCarryingUpdown2		 :UINT :=25;	//1号叠台	负极搬运升降凸轮从叠台位到取料位
P2M1CaDTCarryingUpDown1		 :UINT :=26;	//1号叠台	负极叠台搬运升降凸轮从取料位到叠台位
P2M1CaDTCarryingUpDown2		 :UINT :=27;	//1号叠台	负极叠台搬运升降凸轮从叠台位到取料位
P2M1LeftYDUpdown		 :UINT :=28;	//1号叠台	左压刀升降
P2M1LeftYDLine		 :UINT :=29;	//1号叠台	左压刀开合
P2M1RightYDUpdown		 :UINT :=30;	//1号叠台	右压刀升降
P2M1RightYDLine		 :UINT :=31;	//1号叠台	右压刀开合
P2M1SEPTATLine1		 :UINT :=32;	//1号叠台	隔膜平移从负极到正极
P2M1SEPTATLine2		 :UINT :=33;	//1号叠台	隔膜平移从正极到负极
P2M1SEPTATCache		 :UINT :=34;	//1号叠台	隔膜缓存
P2M1SEPTAunwinding		 :UINT :=35;	//1号叠台	隔膜放卷
P2M1TailCurlUpDown		 :UINT :=36;	//1号叠台	尾卷夹升降
P2M1TailCurlLine		 :UINT :=37;	//1号叠台	尾卷夹平移
				
				
				
P2M2AnCarryingLine1     	 	 :UINT :=41;	//2号叠台	正极搬运平移凸轮号从取料位到叠台位
P2M2AnCarryingLine2   		 :UINT :=42;	//2号叠台	正极搬运平移凸轮号从叠台位到取料位
P2M2AnDTCarryingLine1		 :UINT :=43;	//2号叠台	正极叠台搬运平移凸轮从取料位到叠台位
P2M2AnDTCarryingLine2		 :UINT :=44;	//2号叠台	正极叠台搬运平移凸轮从叠台位到取料位
P2M2AnCarryingUpdown1		 :UINT :=45;	//2号叠台	正极搬运升降凸轮从取料位到叠台位
P2M2AnCarryingUpdown2		 :UINT :=46;	//2号叠台	正极搬运升降凸轮从叠台位到取料位
P2M2AnDTCarryingUpDown1		 :UINT :=47;	//2号叠台	正极叠台搬运升降凸轮从取料位到叠台位
P2M2AnDTCarryingUpDown2		 :UINT :=48;	//2号叠台	正极叠台搬运升降凸轮从叠台位到取料位
P2M2AnCarryingWhirling1		 :UINT :=49;	//2号叠台	正极搬运旋转凸轮从取料位到叠台位
P2M2AnCarryingWhirling2		 :UINT :=50;	//2号叠台	正极搬运旋转凸轮从叠台位到取片位
P2M2CaCarryingLine1     	 	 :UINT :=51;	//2号叠台	负极搬运平移凸轮号从取料位到叠台位
P2M2CaCarryingLine2   		 :UINT :=52;	//2号叠台	负极搬运平移凸轮号从叠台位到取料位
P2M2CaDTCarryingLine1		 :UINT :=53;	//2号叠台	负极叠台搬运平移凸轮从取料位到叠台位
P2M2CaDTCarryingLine2		 :UINT :=54;	//2号叠台	负极叠台搬运平移凸轮从叠台位到取料位
P2M2CaCarryingUpdown1		 :UINT :=55;	//2号叠台	负极搬运升降凸轮从取料位到叠台位
P2M2CaCarryingUpdown2		 :UINT :=56;	//2号叠台	负极搬运升降凸轮从叠台位到取料位
P2M2CaDTCarryingUpDown1		 :UINT :=57;	//2号叠台	负极叠台搬运升降凸轮从取料位到叠台位
P2M2CaDTCarryingUpDown2		 :UINT :=58;	//2号叠台	负极叠台搬运升降凸轮从叠台位到取料位
P2M2LeftYDUpdown		 :UINT :=59;	//2号叠台	左压刀升降
P2M2LeftYDLine		 :UINT :=60;	//2号叠台	左压刀开合
P2M2RightYDUpdown		 :UINT :=61;	//2号叠台	右压刀升降
P2M2RightYDLine		 :UINT :=62;	//2号叠台	右压刀开合
P2M2SEPTATLine1		 :UINT :=63;	//2号叠台	隔膜平移从负极到正极
P2M2SEPTATLine2		 :UINT :=64;	//2号叠台	隔膜平移从正极到负极
P2M2SEPTATCache		 :UINT :=65;	//2号叠台	隔膜缓存
P2M2SEPTAunwinding		 :UINT :=66;	//2号叠台	隔膜放卷
P2M2TailCurlUpDown		 :UINT :=67;	//2号叠台	尾卷夹升降
P2M2TailCurlLine		 :UINT :=68;	//2号叠台	尾卷夹平移
				
				
				
P2M3AnCarryingLine1     	 	 :UINT :=72;	//3号叠台	正极搬运平移凸轮号从取料位到叠台位
P2M3AnCarryingLine2   		 :UINT :=73;	//3号叠台	正极搬运平移凸轮号从叠台位到取料位
P2M3AnDTCarryingLine1		 :UINT :=74;	//3号叠台	正极叠台搬运平移凸轮从取料位到叠台位
P2M3AnDTCarryingLine2		 :UINT :=75;	//3号叠台	正极叠台搬运平移凸轮从叠台位到取料位
P2M3AnCarryingUpdown1		 :UINT :=76;	//3号叠台	正极搬运升降凸轮从取料位到叠台位
P2M3AnCarryingUpdown2		 :UINT :=77;	//3号叠台	正极搬运升降凸轮从叠台位到取料位
P2M3AnDTCarryingUpDown1		 :UINT :=78;	//3号叠台	正极叠台搬运升降凸轮从取料位到叠台位
P2M3AnDTCarryingUpDown2		 :UINT :=79;	//3号叠台	正极叠台搬运升降凸轮从叠台位到取料位
P2M3AnCarryingWhirling1		 :UINT :=80;	//3号叠台	正极搬运旋转凸轮从取料位到叠台位
P2M3AnCarryingWhirling2		 :UINT :=81;	//3号叠台	正极搬运旋转凸轮从叠台位到取片位
P2M3CaCarryingLine1     	 	 :UINT :=82;	//3号叠台	负极搬运平移凸轮号从取料位到叠台位
P2M3CaCarryingLine2   		 :UINT :=83;	//3号叠台	负极搬运平移凸轮号从叠台位到取料位
P2M3CaDTCarryingLine1		 :UINT :=84;	//3号叠台	负极叠台搬运平移凸轮从取料位到叠台位
P2M3CaDTCarryingLine2		 :UINT :=85;	//3号叠台	负极叠台搬运平移凸轮从叠台位到取料位
P2M3CaCarryingUpdown1		 :UINT :=86;	//3号叠台	负极搬运升降凸轮从取料位到叠台位
P2M3CaCarryingUpdown2		 :UINT :=87;	//3号叠台	负极搬运升降凸轮从叠台位到取料位
P2M3CaDTCarryingUpDown1		 :UINT :=88;	//3号叠台	负极叠台搬运升降凸轮从取料位到叠台位
P2M3CaDTCarryingUpDown2		 :UINT :=89;	//3号叠台	负极叠台搬运升降凸轮从叠台位到取料位
P2M3LeftYDUpdown		 :UINT :=90;	//3号叠台	左压刀升降
P2M3LeftYDLine		 :UINT :=91;	//3号叠台	左压刀开合
P2M3RightYDUpdown		 :UINT :=92;	//3号叠台	右压刀升降
P2M3RightYDLine		 :UINT :=93;	//3号叠台	右压刀开合
P2M3SEPTATLine1		 :UINT :=94;	//3号叠台	隔膜平移从负极到正极
P2M3SEPTATLine2		 :UINT :=95;	//3号叠台	隔膜平移从正极到负极
P2M3SEPTATCache		 :UINT :=96;	//3号叠台	隔膜缓存
P2M3SEPTAunwinding		 :UINT :=97;	//3号叠台	隔膜放卷
P2M3TailCurlUpDown		 :UINT :=98;	//3号叠台	尾卷夹升降
P2M3TailCurlLine		 :UINT :=99;	//3号叠台	尾卷夹平移

*)

END_STRUCT
END_TYPE

// ---- P2DUTs/31_其他辅助/DToM_Process.TcDUT
TYPE DToM_Process ://叠片→模切  生产过程数据
STRUCT
	bAn_M1Done:BOOL;//1号叠台正极取料完成
	bAn_M2Done:BOOL;//2号叠台正极取料完成
	bAn_M3Done:BOOL;//3号叠台正极取料完成
	
	bAn_M1Safety:BOOL;//1号叠台正极安全(取料运行时:=FALSE)
	bAn_M2Safety:BOOL;//2号叠台正极安全(取料运行时:=FALSE)
	bAn_M3Safety:BOOL;//3号叠台正极安全(取料运行时:=FALSE)
	
	bCa_M1Done:BOOL;//1号叠台负极取料完成
	bCa_M2Done:BOOL;//2号叠台负极取料完成
	bCa_M3Done:BOOL;//3号叠台负极取料完成
	
	bCa_M1Safety:BOOL;//1号叠台负极安全(取料运行时:=FALSE)
	bCa_M2Safety:BOOL;//2号叠台负极安全(取料运行时:=FALSE)
	bCa_M3Safety:BOOL;//3号叠台负极安全(取料运行时:=FALSE)	
	
	
	bAn_M1LockReady:BOOL;//1号叠台正极锁定准备好
	bAn_M2LockReady:BOOL;//2号叠台正极锁定准备好
	bAn_M3LockReady:BOOL;//3号叠台正极锁定准备好
		
	bCa_M1LockReady:BOOL;//1号叠台负极锁定准备好
	bCa_M2LockReady:BOOL;//2号叠台负极锁定准备好
	bCa_M3LockReady:BOOL;//3号叠台负极锁定准备好

	bAn_M1JumpReady:BOOL;//1号叠台正极锁定 未准备好
	bAn_M2JumpReady:BOOL;//2号叠台正极锁定 未准备好
	bAn_M3JumpReady:BOOL;//3号叠台正极锁定 未准备好
		
	bCa_M1JumpReady:BOOL;//1号叠台负极锁定 未准备好
	bCa_M2JumpReady:BOOL;//2号叠台负极锁定 未准备好
	bCa_M3JumpReady:BOOL;//3号叠台负极锁定 未准备好	
	
	bAn_M1LockingCancel:BOOL;//叠台1锁定中取消
	bAn_M2LockingCancel:BOOL;//叠台2锁定中取消
	bAn_M3LockingCancel:BOOL;//叠台3锁定中取消
	
	bCa_M1LockingCancel:BOOL;//叠台1锁定中取消
	bCa_M2LockingCancel:BOOL;//叠台2锁定中取消
	bCa_M3LockingCancel:BOOL;//叠台3锁定中取消	
	
	bAn_M1PoleHave:BOOL;//叠台1正极取料位无片
	bAn_M2PoleHave:BOOL;//叠台2正极取料位无片
	bAn_M3PoleHave:BOOL;//叠台3正极取料位无片
	
	bCa_M1PoleHave:BOOL;//叠台1负极取料位无片
	bCa_M2PoleHave:BOOL;//叠台2负极取料位无片
	bCa_M3PoleHave:BOOL;//叠台3负极取料位无片
	

END_STRUCT
END_TYPE

// ---- P2DUTs/31_其他辅助/DToM_System.TcDUT
TYPE DToM_System ://叠片→模切  系统数据
STRUCT
	bP2M1Enable:BOOL;//TRUE 1号叠片启用
	bP2M2Enable:BOOL;//TRUE 2号叠片启用
	bP2M3Enable:BOOL;//TRUE 3号叠片启用
	
	bP2Estop:BOOL;//TRUE 叠片急停
	bP2Start:BOOL;//TRUE 叠片启动
	bP2Runing:BOOL;//TRUE 叠片自动中
	
//清尾料
	bP2ClearDo:BOOL;//叠片开始清尾料   注：先发需求量，再发清尾料开始信号
	iAn1Ask:INT:=0;// 1号正极极片需求量
	iAn2Ask:INT:=0;// 2号正极极片需求量
	iAn3Ask:INT:=0;// 3号正极极片需求量
	iCa1Ask:INT:=0;// 1号负极极片需求量
	iCa2Ask:INT:=0;// 2号负极极片需求量
	iCa3Ask:INT:=0;// 3号负极极片需求量
	bP2ClearDone:BOOL;//叠片清尾料完成	
	
//光电信号传递
	bAnBelt1Have:BOOL;//正极分段皮带1有料感应
	bAnBelt2Have:BOOL;//正极分段皮带2有料感应
	bAnBelt3Have:BOOL;//正极分段皮带3有料感应
	bCaBelt1Have:BOOL;//负极分段皮带1有料感应
	bCaBelt2Have:BOOL;//负极分段皮带2有料感应
	bCaBelt3Have:BOOL;//负极分段皮带3有料感应
	
	P3SaveParDone      :BOOL;//p3保存参数完成
	P3ReadParDone     :BOOL;//p3读取参数完成
	
	fM1MainSetPos:REAL;//叠片1主轴指令位置
	fM2MainSetPos:REAL;//叠片2主轴指令位置
	fM3MainSetPos:REAL;//叠片3主轴指令位置
END_STRUCT
END_TYPE

// ---- P2DUTs/31_其他辅助/File_com_typ.TcDUT
TYPE File_com_typ :(*xml内部用*)
STRUCT
	FileName_save: 		T_MaxString	 := 'test.xml';		(* File name would be saved setting by the HMI用来保存的文件名称 *)
	FileName_active: 	T_MaxString	 := 'test.xml';		(* File name activated now to be loaded 用来读取的文件目标文件名*)
	Device: 			T_MaxString  := '\Hard Disk\';		(* Device: C:\ or USB    or ce   \Hard Disk\*)
	DeviceNum:		INT:=3;							(* 1= C:\ or 2=USB    or 3= ce   \Hard Disk\*)
	Var_Name: 			ARRAY [0..19] OF T_MaxString;	(* Variable name which need to be loaded or saved *)
	Dir_change:			BOOL;							(* Command for change the directory	*)
	File_load:			BOOL;							(* Command for load the exiting file	*)
	File_save:			BOOL;							(* Command for save the file	*)
	File_del:			BOOL;							(* Command for delete the exiting file	*)
	File_copy:			BOOL;							(* Command for copy the exiting file between the C:\ and USB *)
	Err_ack:			BOOL;							(* Command for acklonege the error	*)
	bBusy:				BOOL;							(* State for the FB running	*)
	ErrorID:			UDINT;							(* Error ID from the FB *)
END_STRUCT
END_TYPE

// ---- P2DUTs/31_其他辅助/MToD_Process.TcDUT
TYPE MToD_Process ://模切→叠片  生产过程数据
STRUCT
	bAn_M1Allow:BOOL;//允许1号叠台正极取料
	bAn_M2Allow:BOOL;//允许2号叠台正极取料
	bAn_M3Allow:BOOL;//允许3号叠台正极取料

	bAn_M1Allow2:BOOL;//允许1号叠台正极取料
	bAn_M2Allow2:BOOL;//允许2号叠台正极取料
	bAn_M3Allow2:BOOL;//允许3号叠台正极取料
	
	bCa_M1Allow:BOOL;//允许1号叠台负极取料
	bCa_M2Allow:BOOL;//允许2号叠台负极取料
	bCa_M3Allow:BOOL;//允许3号叠台负极取料	
	
	bCa_M1Allow2:BOOL;//允许1号叠台负极取料
	bCa_M2Allow2:BOOL;//允许2号叠台负极取料
	bCa_M3Allow2:BOOL;//允许3号叠台负极取料		
	
	bAn_M1Locking:BOOL;//叠台1锁定中
	bAn_M2Locking:BOOL;//叠台2锁定中
	bAn_M3Locking:BOOL;//叠台3锁定中
	
	bCa_M1Locking:BOOL;//叠台1锁定中
	bCa_M2Locking:BOOL;//叠台2锁定中
	bCa_M3Locking:BOOL;//叠台3锁定中
END_STRUCT
END_TYPE

// ---- P2DUTs/31_其他辅助/MToD_System.TcDUT
TYPE MToD_System ://模切→叠片  系统数据
STRUCT
	bP1Estop:BOOL;//TRUE 模切急停
	bP1Start:BOOL;//TRUE 模切启动
	bP1Runing:BOOL;//TRUE 模切自动中
	iCarryPoleMode:INT:=3;//极片仅流至1.2.3工位
	p1state:INT;//模切状态 1:自动中   2:自动-Ready  3:手动   4:急停    5：报警    6.自动-NoReady
	P1SaveParDone      :BOOL;//模切保存参数完成
	P1ReadParDone     :BOOL;//模切读取参数完成
//清尾料
	bP1ClearDo:BOOL;//模切开始清尾料   注：模切部分程序必须在叠片开始清尾料后，在进入清尾料流程
	bP1ClearDone:BOOL;//模切清尾料完成	注：必须叠台部分叠完所有极片立马给模切 叠片清尾料完成，最后模切反馈清尾料完成
END_STRUCT
END_TYPE

// ---- P2DUTs/31_其他辅助/ST_DATA_NEED_BE_PERSIS.TcDUT
TYPE ST_DATA_NEED_BE_PERSIS :(*需要断电保持的参数*)(*中间变量，只用在判断用*)
STRUCT

	strSetLevelPassword: 	ARRAY [0..3] OF STRING(80) := ['0','1','2','3'];
	strInputReceipeName: 	STRING(80);
	strCurrentReceipeName: 	STRING(80);

END_STRUCT
END_TYPE

// ---- P2DUTs/32_系统/IModeEN.TcDUT
TYPE IModeEN ://功能屏蔽
STRUCT

	FirstEmpFoldEN		:BOOL;  		// 首层空叠隔膜屏蔽   ON是屏蔽
	DP_ModeEN			:BOOL;		//尾层空叠隔膜屏蔽	OFF是屏蔽
	RectifydevModelEN		:BOOL;		//隔膜纠偏屏蔽		ON是屏蔽
	EmptyRunModeEN		:BOOL;		//空叠隔膜屏蔽		OFF是屏蔽
	CCD_ChosesHMIEN		:BOOL;		//CCD屏蔽		ON是屏蔽
	DT_CCD_TwoModelEN	:BOOL;		//CCD复检屏蔽		ON是屏蔽
	DT_OverhangEN		:BOOL;		//对齐度屏蔽		ON是屏蔽
	DT_CellNG_TFEN		:BOOL;		//对齐度踢废屏蔽 	ON是屏蔽
	DT_OHclosureEN		:BOOL;		//对齐度闭环屏蔽		ON是屏蔽
	GMAngleALMsel     :BOOL;		//隔膜卷径报警屏蔽		ON是屏蔽
END_STRUCT
END_TYPE

// ---- P2DUTs/32_系统/IRecipe.TcDUT
TYPE IRecipe :
STRUCT
	bCreate:BOOL;
	bSave:BOOL;
	bLoad:BOOL;

     
END_STRUCT
END_TYPE

// ---- P2DUTs/32_系统/ST_SysCmd.TcDUT
TYPE ST_SysCmd :
STRUCT

(*主页面指令*)
	bInit							:BOOL;	(*初始化*)

	bShutDownPc					:BOOL;	(*关机，程序做延迟*)
	bRebootPc						:BOOL;	(*重启PC*)
	bSaveData						:BOOL;	(*保存所有参数*)
    bReadData						:BOOL;	(*读取所有参数*)


END_STRUCT
END_TYPE

// ---- P2DUTs/32_系统/ST_SystemRUN.TcDUT
TYPE ST_SystemRUN ://系统功能块UDT
STRUCT
(***btn***)
	 btnStart                      :BOOL;  
     btnStop                      :BOOL;   
	 btnReset                     :BOOL;  
     btnAuto                      :BOOL;
     btnManul                   :BOOL;	 
	 btnEstop                    :BOOL;
	// btnDoor: ARRAY[1..10] OF BOOL;//门禁
	  bReset                      :BOOL;  
(***HMI*) 
	 hmiStart                    :BOOL;  
     hmiStop                    :BOOL;   
	 hmiReset                   :BOOL;  
     hmiAutoSwitch           :BOOL;
     hmiAuto                    :BOOL;
     hmiManul                  :BOOL;	 
	 hmiEstop                   :BOOL;
     hmiTest                     :BOOL;
(**Status**)
	 FlgAuto                     :BOOL;       //自动中标志位 硬件状态
	 FlgManua                  :BOOL;      //手动状态硬件状态
     iMode                       :INT;  //运行模式  1:自动中   2:暂停  3:手动   4:急停   

     Autoing                     :BOOL;   //自动运行中
	 Manuling                   :BOOL;  //手动运行中
	 Stoping                     :BOOL;   //停止中
	 Alarming                   :BOOL;   //报警中
	 bErrorStop                :BOOL;//报警停机

     bAutoCondition         :BOOL;
     bStopFinished            :BOOL;
 
//凸轮初始化
   // bP2M1Init                   :BOOL;
   // bP2M2Init                   :BOOL;
   // bP2M3Init                  :BOOL;
    //bP2M1InitDone              :BOOL;
   // bP2M2InitDone               :BOOL;
 //   bP2M3InitDone               :BOOL;
    bInitDone              :BOOL;	
	TheFirstTimebool     :BOOL;//第一次上电标志
	bwindow	          :BOOL;  // 弹窗  
	bccdstate        :BOOL;  //CCD状态
END_STRUCT
END_TYPE

// ---- P2DUTs/33_M2/ST_BeltData.TcDUT
TYPE ST_BeltData :
STRUCT
 	bHavePole   								:		 BOOL		 ;//		是否有极片
 	iPanoramaNG									:		 INT		 ;//		尺寸检测状态  1:OK  2:NG   3:无极片    0:无效
 	iJumpCutNG									:		 INT		 ;//		跳切连续NG  1:OK  2:NG  0:无效
 	fPoleWidth									:		 REAL		 ;//		片宽
  	fPoleHeigh									:		 REAL		 ;//		片高
  	stPoleNo									:		 STRING(256) ;//		模切极片编号
 // fbST_CCDComSize								:		 ST_CCDComSize;
	fTabWidth									:		 REAL		 ;//		尺寸检测CCD结果(极耳宽度)
	fTabHeigh									:		 REAL		 ;//		尺寸检测CCD结果(极耳高度)
	fTabSite   									: 		 REAL		 ;// 		极耳左，右边距(就是极耳位置，不分左右)
	//fOffsetDeg								:		 REAL		 ;//		尺寸检测CCD结果(极片裁切面角度偏移)
	RoundedSize1                                :        REAL        ;//        圆角尺寸1纵深
	RoundedSize2                                :        REAL        ;//        圆角尺寸2纵深
	RoundedSize3                                :        REAL        ;//        圆角尺寸3纵深
	RoundedSize4                                :        REAL        ;//        圆角尺寸4纵深
	RoundedSize5                                :        REAL        ;//        圆角尺寸5横深
	RoundedSize6                                :        REAL        ;//        圆角尺寸6横深
	RoundedSize7                                :        REAL        ;//        圆角尺寸7横深
	RoundedSize8                               	:        REAL        ;//        圆角尺寸8横深
	PolePlateAngle1                             :        REAL        ;//        极片角度1  极片角度
	PolePlateAngle2                             :        REAL        ;//        极片角度2
	PolePlateAngle3                             :        REAL        ;//        极片角度3
	PolePlateAngle4                             :        REAL        ;//        极片角度4
	fPoleNGSizeNo								:		 REAL		 ;//		尺寸检测CCD结果(NG分类编号)
	iTabNGSizeNo:INT;  //尺寸检测CCD极耳抓边异常分类     1： OK  2: 极片抓边异常    3:极耳抓边异常     4：都抓边异常     5：极片或极耳角度异常    
	
	iPoleRAngleNG								:		 INT		 ;//		尺寸检测CCD结果(R角NG)
	iFinish										:        INT		 ;//		尺寸检测CCD结果指示(1=完成;2=NG;3=无片;0=无效)  SizeResults
	AppearanceResult							:        INT		 ;//	    极片外观判定结果   线扫NG、OK

	UnreelingTension                       	    :        REAL        ;//        放卷张力
	SlicingSpeed                                :        REAL        ;//        切片速度
	PolePlateLenth                              :        REAL        ;//        极片长度（走带方向）
	fPoleNGSacnNo:REAL;  //极片先扫NG编号(NG分类编号)	
	
	bYellowMark:BOOL;//黄标标志--TRUE为黄标
	bBlueMark:BOOL;//接带标志--TRUE为接带
	Code			:STRING(49);//料卷条码
END_STRUCT
END_TYPE

// ---- P2DUTs/33_M2/ST_BeltData1.TcDUT
TYPE ST_BeltData1 ://皮带NG数据
STRUCT
	
  bHavePole   :BOOL;  //是否有极片

  iPanoramaNG:INT;//尺寸检测状态  1:OK  2:NG   3:无极片    0:无效
  
  iLineScanUpNG:INT;//线扫上  1:OK  2:NG  0:无效
  
  iLineScanDownNG:INT;//线扫下  1:OK  2:NG     0:无效
  
  iYellowNG: INT;//黄标NG  0:OK   1:NG 
  
END_STRUCT
END_TYPE

// ---- P2DUTs/34_M1/ST_Rectify.TcDUT
TYPE ST_Rectify :   //纠偏控制
STRUCT
(********参数**************)	

	bReset            :BOOL;     // 纠偏复位  
	bEnable		:BOOL;	(*开启自动纠偏*)
	fSensorActValue			:REAL; //实际位置
	
	bReady              :BOOL;  //纠偏准备号
	bAutoRunning		:BOOL;	(*纠偏自动运行中*)
	Error		:BOOL;            //纠偏错误
    ErrID:	 STRING;     //纠偏错误代码
	
END_STRUCT
END_TYPE

// ---- P2DUTs/35_CCD/35_CCD/ICCD_1.TcDUT
TYPE ICCD_1 : 
STRUCT
	bComOpen:BOOL;  //扫码Tcp 开
    bComClose:BOOL;  //扫码Tcp 关

	bSend :BOOL; //  扫码开
	//bLOFF :BOOL; //扫码关
	bDone  :BOOL; //扫码完成
    bError :BOOL;//扫码故障	
    strReceive:STRING;//

END_STRUCT
END_TYPE

// ---- P2DUTs/35_CCD/35_CCD/STCcdData_1.TcDUT
TYPE STCcdData_1 :
STRUCT
	iorder:DINT;  //功能码  2  3   4    
	strCode:STRING   ;//二维码
	strShortData: STRING; //短路测试数据 128
	strBetryName: STRING;//文件名
	strHotPress: STRING;//热压参数
END_STRUCT
END_TYPE

// ---- P2DUTs/35_CCD/35_CCD/ST_CCDCom.TcDUT
TYPE ST_CCDCom : 
STRUCT
	bHeartbeat :BOOL;  //叠片部分ccd软件心跳
	
	AnRec:ST_CCDComRectify;//正极纠偏工位
	CaRec:ST_CCDComRectify;//负极纠偏工位
	Over:ST_CCDComOverhang;//对齐度工位
END_STRUCT
END_TYPE

// ---- P2DUTs/35_CCD/35_CCD/ST_CCDComOverhang.TcDUT
TYPE ST_CCDComOverhang :
STRUCT
	Start:ST_CCDOverhang_O;  //软触发
	Finish:ST_CCDOverhang_I;  //检测结果
	bRectifyDone:BOOL;  //取图完成
END_STRUCT
END_TYPE

// ---- P2DUTs/35_CCD/35_CCD/ST_CCDComRectify.TcDUT
TYPE ST_CCDComRectify :
STRUCT
	Start:ST_CCDComRectify_O;  //软触发
	Finish:ST_CCDComRectify_I;  //纠偏结果
	DayNgclassification :ST_Ng_classification; //白班纠偏NG计数
	NightNgclassification :ST_Ng_classification; //晚班纠偏NG计数
	bRectifyDone:BOOL;  //取图完成
	iDemarcatResult:INT;//标定结果（1:OK ,2:NG,3:无料）
	iDemCount:INT;//标定拍照计数


END_STRUCT
END_TYPE

// ---- P2DUTs/35_CCD/35_CCD/ST_CCDComRectify_I.TcDUT
TYPE ST_CCDComRectify_I :
STRUCT
	
	NG_Code:INT;     //  NG代码
	RectifyX1:REAL;  //纠偏平台X1方向纠偏量
	RectifyX2:REAL;  //纠偏平台X2方向纠偏量
	RectifyY:REAL;  //纠偏平台Y方向纠偏量
	RectifyResult:INT;//纠偏结果（1:OK ,2:NG,3:无料 4:纠偏结果NG）
	Offset_X: REAL;//OH闭环计算偏移值X
	Offset_Y: REAL;//OH闭环计算偏移值Y
END_STRUCT
END_TYPE

// ---- P2DUTs/35_CCD/35_CCD/ST_CCDComRectify_O.TcDUT
TYPE ST_CCDComRectify_O :
STRUCT
	iPhotoDo:INT;//拍照软触发,1=正常纠偏拍照，2=复检，3=有无片拍照（全视野）     4.有无片报警拍照（检测四角)
	PhotoFinish:INT;//叠台电芯最后一片标记
	stPoleNo:STRING(256);  //极片编号

	
END_STRUCT
END_TYPE

// ---- P2DUTs/35_CCD/35_CCD/ST_CCDOverhang_I.TcDUT
TYPE ST_CCDOverhang_I :
STRUCT
	OverhandResult	:	INT	    ;// 对齐度结果（1:OK ,2:NG,3:无料 4:极耳顶宽NG）
	OverhandiPliesNo:   INT     ;// 返回极片层数
	PoleOverhandX1	:	REAL	;//	极片与隔膜X1
	PoleOverhandY1	:	REAL	;//	极片与隔膜Y1
	PoleOverhandX2	:	REAL    ;// 极片与隔膜X2
	PoleOverhandY2	:	REAL    ;// 极片与隔膜Y2
	PoleOverhandX3	:	REAL    ;// 极片与隔膜X3
	PoleOverhandY3	:	REAL    ;// 极片与隔膜Y3
	PoleOverhandX4	:	REAL	;//	极片与隔膜X4
	PoleOverhandY4	:	REAL	;//	极片与隔膜Y4
	AnCaOverhandX1	:	REAL	;//	负极与正极X1
	AnCaOverhandY1	:	REAL	;//	负极与正极Y1
	AnCaOverhandX2	:	REAL	;// 负极与正极X2
	AnCaOverhandY2	:	REAL	;//	负极与正极Y2
	AnCaOverhandX3	:	REAL	;// 负极与正极X3
	AnCaOverhandY3	:	REAL	;//	负极与正极Y3
	AnCaOverhandX4	:	REAL	;// 负极与正极X4
	AnCaOverhandY4	:	REAL	;//	负极与正极Y4
	AddOverhangX1	:	REAL	;//	极片整体对齐度X1
	AddOverhangY1	:	REAL	;//	极片整体对齐度Y1
	AddOverhangX2	:	REAL	;//	极片整体对齐度X2
	AddOverhangY2	:	REAL	;// 极片整体对齐度Y2
	AddOverhangX3	:	REAL	;//	极片整体对齐度X3
	AddOverhangY3	:	REAL	;// 极片整体对齐度Y3
	AddOverhangX4	:	REAL	;//	极片整体对齐度X4
	AddOverhangY4	:	REAL	;//	极片整体对齐度Y4
	OverhangXY_Warm	:	INT		;//连续10片对齐度超限报警	
	stCellNo		:	STRING(256);//电芯编号	
END_STRUCT
END_TYPE

// ---- P2DUTs/35_CCD/35_CCD/ST_CCDOverhang_O.TcDUT
TYPE ST_CCDOverhang_O :
STRUCT
	iPhotoDo:INT;//1为正常对齐度拍照，2为叠台检测有无拍照
	iPliesNo:INT;  //当前层数
	OverhangXY_Warm_Reset : INT; //超限预警返回值
	stPoleNo:STRING(256);  //极片编号
	
	
END_STRUCT
END_TYPE

// ---- P2DUTs/35_CCD/35_CCD/ST_Ng_classification.TcDUT
TYPE ST_Ng_classification :
STRUCT
	X1_NG    :UINT;//X1纠偏不良数
    X2_NG    :UINT;//X2纠偏不良数
    Y_NG    :UINT;//Y纠偏不良数
    R_NG    :UINT;//R角轮廓不良数
    other_NG    :UINT;//其他类不良数
	NgClear     :ARRAY [1..6] OF BOOL ;//不良数清零
	
END_STRUCT
END_TYPE

// ---- P2DUTs/35_CCD/ICCD.TcDUT
TYPE ICCD : 
STRUCT
	bComOpen:BOOL;  //扫码Tcp 开
    bComClose:BOOL;  //扫码Tcp 关

	bSend :BOOL; //  扫码开
	//bLOFF :BOOL; //扫码关
	bDone  :BOOL; //扫码完成
    bError :BOOL;//扫码故障	
    strReceive:STRING;//

END_STRUCT
END_TYPE

// ---- P2DUTs/35_CCD/STCcdData.TcDUT
TYPE STCcdData :
STRUCT
	iorder:DINT;  //功能码  2  3   4    
	strCode:STRING   ;//二维码
	strShortData: STRING; //短路测试数据 128
	strBetryName: STRING;//文件名
	strHotPress: STRING;//热压参数
END_STRUCT
END_TYPE

// ---- P2DUTs/35_CCD/STCcdDataSend.TcDUT
TYPE STCcdDataSend :
STRUCT
	iHead :DINT:=32767;
	iorder:DINT:=2;
	strCode:ARRAY[0..63] OF   BYTE    ;//二维码
	strShortData: ARRAY[0..127] OF BYTE; //短路测试数据 128
	strBetryName: ARRAY[0..31] OF BYTE;//文件名
	strHotPress: ARRAY[0..63] OF BYTE;//热压参数
    iEnd :DINT:=65535;
END_STRUCT
END_TYPE

// ---- P2DUTs/36_ShortTest/CMD.TcDUT
TYPE CMD :
STRUCT
	RST :                   STRING:='*RST';     // 1 仪器初始化
    Start :                 STRING:=':STARt';// 2 测试开始
    Stop :                  STRING:=':STOP';// 3  测试停止
    State_Check :           STRING:=':STATe?';// 4 测试状态查询 0：停止中  1：测试中   2：放电中
	
    Measure_Check :         STRING:=':MEASure?';// 5  测量值查询
    Measure_Check2 :        STRING:=':MEASure:RESult?';// 6  测量值，判定结果查询  //1:OFF 2:NOcomp 3:DELAY 4:PASS 5:UFAIL 6:LFAIL 7:ULFA
    Measure_Clear :         STRING:=':MEASure:CLEar';// 7  测量值，判定结果清除
	
    Voltage :               STRING:=':VOLTage';// 8  测试电压设置
    Voltage_Check :         STRING:=':VOLTage?';// 9  测试电压查询 
    Voltage_Monitor :       STRING:=':MEASure:MONItor?';// 10  电压值监视
	
    Mohm_Range :            STRING:=':MOHM:RANGe';// 11  电阻量程设置(2M/20M/200M/2000M/4000M/AUTO)  
    Mohm_Range_Check :      STRING:=':MOHM:RANGe?';// 12  电阻量程查询
	
    Speed :                 STRING:=':SPEed';// 13 测量速度设置(FAST/SLOW)
    Speed_Check :           STRING:=':SPEed?';// 14 测量速度查询
	
    Timer :                 STRING:=':TIMer';// 15  测试时间设置
    Timer_Check :           STRING:=':TIMer?';// 16  测试时间查询
    Delay :                 STRING:=':DELay';// 17  响应时间设置(0为自动)
    Delay_Check :           STRING:=':DELay?';// 18  响应时间查询(0为自动)
	
    ComparatorLimit :       STRING:=':COMParator:LIMit';// 19  比较器上下限值设置（上限,下限）
    ComparatorLimit_Check : STRING:=':COMParator:LIMit?';// 20  比较器上下限值查询
    ComparatorMode :        STRING:=':COMParator:MODE';// 21  测试模式设置（CONTinue/PASSstop/FAILstop/SEQuence）  
    ComparatorMode_Check :  STRING:=':COMParator:MODE?';// 22 测试模式查询（CONTINUE/PASSSTOP/FAILSTOP/SEQUENCE）
    ComparatorBeeper :      STRING:=':COMParator:BEEPer';// 23  判定蜂鸣器设置(PASS/FAIL/OFF/END)
    ComparatorBeeper_Check :STRING:=':COMParator:BEEPer?';// 24  判定蜂鸣器查询(PASS/FAIL/OFF/END)
	
    Contact :               STRING:=':CONTactcheck';//  25  接触检查功能设置(ON/OFF)	
	Contact_Check :         STRING:=':CONTactcheck?';// 26  接触检查功能查询(ON/OFF)
    Contact_Result :        STRING:=':CONTactcheck:RESult?';// 27  接触检查结果查询(NOCHK/PASS/HFAIL/LFAIL/HLFAIL)
	
    Short :                 STRING:=':SHORtcheck';// 28  短路检查功能设置(ON/OFF)	
    Short_Check :           STRING:=':SHORtcheck?';// 29  短路检查功能查询 
    ShortTime :             STRING:=':SHORtcheck:TIME';// 30 短路检查时间设置(0:自动)
    ShortTime_Check :       STRING:=':SHORtcheck:TIME?';// 31  短路检查时间查询
    Short_Result :          STRING:=':SHORtcheck:RESult?';// 32  短路检查结果查询（NOCHK/PASS/FAIL）
	
    KeyBeeper :             STRING:=':KEY:BEEPer';// 33  按键输入蜂鸣器音设置(ON/OFF)	
    KeyBeeper_Check :       STRING:=':KEY:BEEPer?';// 34  按键输入蜂鸣器音查询
   
END_STRUCT
END_TYPE

// ---- P2DUTs/36_ShortTest/IShortTest.TcDUT
TYPE IShortTest : 
STRUCT
	bStart :BOOL; //
	bDone  :BOOL; //

   iResult:INT; // 1 OK  2 NG
    
   ErrorID :INT;
   
	

END_STRUCT
END_TYPE

// ---- P2DUTs/36_ShortTest/ShortDataShow.TcDUT
TYPE ShortDataShow :
STRUCT
	strState:STRING;         //0：停止中  1：测试中   2：放电中
    strResult:STRING;  //启动测试后返回结果   综合结果
	
	strMeasure :STRING;     //测量电阻值
	strMeasureState :STRING;     //1:OFF 2:NOcomp 3:DELAY 4:PASS 5:UFAIL 6:LFAIL 7:ULFAIL

	strVoltageSetValue:STRING;  //电压设定值查询
    strVoltageMonitor:STRING; //电压值监视
	
	strMohmRangeValue:STRING;//(1:2M/2:20M/3:200M/4:2000M/5:4000M/6:AUTO) 
    
	strSpeedValue:STRING ;//测量速度查询(FAST/SLOW)
	
	strTimerValue :STRING;  //测试时间查询
	strDelayValue :STRING;  //响应时间查询(0自动）
	
	strComparatorLimitSet :STRING;  //比较器上限 下限值
	strComparatorModeValue: STRING ;// 21  测试模式查询（CONTinue/PASSstop/FAILstop/SEQuence）
	strComparatorBeeperValue:    STRING;//23  判定蜂鸣器查询(PASS/FAIL/OFF/END)
	
	strContactValue :STRING;//  25  接触检查功能查询(ON/OFF)
	strContactResult :STRING;//  27  接触检查结果查询(NOCHK/PASS/HFAIL/LFAIL/HLFAIL)
	
	strShortValue:STRING;// 28  短路检查功能查询(ON/OFF)
	strShortTimeValue:  STRING;// 30 短路检查时间查询(0:自动)
	strShortResult:STRING;// 32  短路检查结果查询（NOCHK/PASS/FAIL）
	
	strKeyBeeperValue:STRING;  // 33  按键输入蜂鸣器音查询(ON/OFF)	

END_STRUCT
END_TYPE

// ---- P2DUTs/36_ShortTest/ShortPar.TcDUT
TYPE ShortPar :
STRUCT
	fVoltageSet: REAL;  //电压设定值

	StrMohmRangeSet:STRING; //电阻量程设置(1:2M/2:20M/3:200M/4:2000M/5:4000M/6:AUTO) 

    StrSpeedSet:STRING ;//测量速度设置(FAST/SLOW)
    
    fTimerSet:    REAL; //测试时间设置
    fDelaySet:   REAL; //响应时间设定
     
	fComparatorUpLimitSet :REAL;  //比较器上限设定
	fComparatorDownLimitSet :REAL;//比较器下限设定	
    strComparatorModeSet: STRING ;// 21  测试模式设置（CONTinue/PASSstop/FAILstop/SEQuence）
	
	strComparatorBeeperSet:    STRING;//23  判定蜂鸣器设置(PASS/FAIL/OFF/END)
	
	strContactSet :STRING;//  25  接触检查功能设置(ON/OFF)	

	strShortSet:STRING;// 28  短路检查功能设置(ON/OFF)
	
	fShortTimeSet:  REAL;// 30 短路检查时间设置(0:自动)
	
	
	strKeyBeeperSet:STRING;  // 33  按键输入蜂鸣器音设置(ON/OFF)	
	
	
END_STRUCT
END_TYPE

// ---- P2DUTs/37_Code/ICode.TcDUT
TYPE ICode : 
STRUCT
	bComOpen                  :BOOL;  //扫码Tcp 开
    bComClose                  :BOOL;  //扫码Tcp 关
 	bComOpenDone          :BOOL;  //扫码Tcp 打开OK
    bCodeConError             :BOOL;//扫码通讯故障

    sRemoteHost                :T_IPv4Addr;  //扫描枪IP地址
    sRemotePot                  :UINT;  //端口号

	bLON                           :BOOL; //  扫码开
	bLOFF                          :BOOL; //扫码关
	bDone                         :BOOL; //扫码完成
    bCodeError                  :BOOL;//扫码故障	
    strCode                       :STRING;//条码结果

END_STRUCT
END_TYPE

// ---- P2DUTs/37_Code/ParCode.TcDUT
TYPE ParCode : 
STRUCT
    sRemoteHost                :T_IPv4Addr;  //扫描枪IP地址
    sRemotePot                  :UINT;  //端口号
    TimeOut:		               INT:=5;	//扫码超时时间


END_STRUCT
END_TYPE

// ---- P2DUTs/38_User1/ControlSignal.TcDUT
TYPE ControlSignal :
STRUCT
	btn:ST_Button;//机架按钮
	se:ST_Senser;//机架信号
	U:ST_UserControl;//用户控制信号
	An_b:conAn_date;//正极取片数据包
	Ca_b:conCa_date;//负极取片数据包
	DT_b:conDT_Date;//叠台数据包
	WJ_b:conTailCurl_date;//尾卷数据包
	TJ_b:conStickGlue_date;//贴胶数据包
	DTRunStatus:conDT_RunStatus;//叠台运行数据	
	
	
END_STRUCT
END_TYPE

// ---- P2DUTs/38_User1/EleControlNo.TcDUT
TYPE EleControlNo ://气缸、真空阀、破真空阀
STRUCT
	CylinderName:ST_CylinderName;//气缸号
	ElectValveName:ST_ElectValveName;//真空和破真空号
END_STRUCT
END_TYPE

// ---- P2DUTs/38_User1/LocalProduction.TcDUT
TYPE  LocalProduction :
STRUCT
	OutFlag1:BOOL;(*产量计数标志1*)
	OutFlag2:BOOL;(*产量计数标志2*)
	NGFlag:ARRAY[1..30] OF BOOL;(*NG1计数标志*)

	RunFlag:BOOL;(*运行标志*)
	WaitFlag:BOOL;(*待料标志*)
	AlarmFlag:BOOL;(*故障标志*)
	DelDataAMBtn:BOOL;(*白班数据清除按钮*)
	DelDataPMBtn:BOOL;(*夜班数据清除按钮*)
	NowOutTotal:REAL;(*当前班次加工总数*)
	NowRate:REAL;(*当前班次良率*)
	HMI_NGClearAMBtn:ARRAY[1..30] OF BOOL;//白班NG类型计数清零
	HMI_NGClearPMBtn:ARRAY[1..30] OF BOOL;//夜班NG类型计数清零
	
//产能清零
	HMI_DelDataAMBtn			:BOOL;//白班产能清零
	HMI_DelDataPMBtn			:BOOL;//夜班产能清零
(*产能统计*)
	HMI_TodayTotal				:REAL;(*当天24H生产总数*)
	HMI_TodayOK					:REAL; (*当天24H生产OK总数*)
	HMI_TodayNG 				:REAL; (*当天24H生产NG总数*)
	
	HMI_HistoryTotal			:ARRAY[1..7 ] 	OF REAL ;(*历史每天24H生产总数ARRAY[1..7 ]*)
	HMI_HistoryOK				:ARRAY[1..7 ] 	OF REAL ;(*历史每天24H生产OK总数ARRAY[1..7 ]*)
	HMI_HistoryNG 				:ARRAY[1..7 ] 	OF REAL ; (*历史每天24H生产NG总数ARRAY[1..7 ]*)
	DayCountTotal				:REAL;(*白班产量合计*)
	NightCountTotal				:REAL;(*夜班产量合计*)
	SaveNowDay					:INT;
	SaveNowMonth				:INT;
	nDayRunTimeCnt				:ARRAY[8..19 ] 	OF UDINT;		(*白班运行时间统计*)
	nDayAlarmTimeCnt			:ARRAY[8..19 ] 	OF UDINT;		(*白班报警时间统计*)
	nDayWaitTimeCnt				:ARRAY[8..19 ] 	OF UDINT;		(*白班待料时间统计*)
	nNightRunTimeCnt			:ARRAY[0..23 ] OF UDINT;		(*夜班运行时间统计*)
	nNightAlarmTimeCnt			:ARRAY[0..23 ] OF UDINT;		(*夜班报警时间统计*)
	nNightWaitTimeCnt			:ARRAY[0..23 ] OF UDINT;		(*夜班待料时间统计*)
	HourTimeDayCount			:ARRAY[8..19 ] 	OF REAL;		(*白班每小时产量*)
	HourTimeNightCount			:ARRAY[0..23] 	OF REAL;		(*夜班每小时产量*)
	NgPerHourDayCount			:ARRAY[1..30 ] 	OF REAL;		(*白班1-30种类的不良分类*)
	NgPerHourNightCount			:ARRAY[1..30 ] 	OF REAL;		(*夜班1-30种类的不良分类*)
	HMI_TotalCount				:REAL;(*总产量*)
	HMI_OkCount					:REAL;(*OK产量*)
	HMI_NgCount					:REAL;(*Ng产量*)
	HMI_Qualified 				:REAL;(*良率*)
	HMI_NG_Qualified 			:REAL;(*不良率*)
	HMI_OEE							:REAL;//设备稼动率
	HMI_DayOkCount				:REAL;(*白班OK产量*)
	HMI_DayNgCount				:REAL;(*白班Ng产量*)
	HMI_DayQualified 			:REAL;(*白班良率*)
	HMI_DayNG_Qualified 		:REAL;(*白班不良率*)
	HMI_NightOkCount			:REAL;(*夜班OK产量*)
	HMI_NightNgCount			:REAL;(*夜班Ng产量*)
	HMI_NightQualified 			:REAL;(*夜班良率*)
	HMI_NightNG_Qualified 		:REAL;(*夜班不良率*)
	DayRunTimeTotal				:REAL;(*白班总运行时间合计*)
	NightRunTimeTotal			:REAL;(*夜班总运行时间合计*)
	DayAlarmTimeTotal			:REAL;(*白班总报警时间合计*)
	NightAlarmTimeTotal			:REAL;(*夜班总报警时间合计*)
	DayWaitTimeTotal			:REAL;(*白班总待料时间合计*)
	NightWaitTimeTotal			:REAL;(*夜班总待料时间合计*)
	RunTimeTotal				:REAL;(*总运行时间合计*)
	WaitTimeTotal				:REAL;(*总待料时间合计*)
	AlarmTimeTotal				:REAL;(*总报警时间合计*)
	(*历史数据变量汇总1-7天*)
	(*白班*)
	DayReadDayHistory			:ARRAY[1..7 ] 	OF INT;(*历史日*)
	DayReadMonthHistory			:ARRAY[1..7 ] 	OF INT;(*历史月*)
	DayCountTotalHistory		:ARRAY[1..7 ] 	OF REAL ;(*历史白班每天生产总数*)
	HMI_DayOkCountHistory		:ARRAY[1..7 ] 	OF REAL ;(*历史白班每天生产OK总数*)
	HMI_DayNgCountHistory		:ARRAY[1..7 ] 	OF REAL ;(*历史白班每天生产NG总数*)
	HMI_DayQualifiedHistory		:ARRAY[1..7 ] 	OF REAL ;  (*历史白班每天良率*)
	DayRunTimeTotalHistory		:ARRAY[1..7 ] 	OF REAL ;(*历史每天白板总运行时间合计*)
	DayWaitTimeTotalHistory		:ARRAY[1..7 ] 	OF REAL ;(*历史每天白板总待料时间合计*)
	DayAlarmTimeTotalHistory	:ARRAY[1..7 ] 	OF REAL ;(*历史每天白板总报警时间合计*)
	NgPerHourDayCountHistory	:ARRAY[1..7,1..30 ] 	OF REAL ;(*历史每天白班各类NG数量*)
	HourTimeDayCountHistory		:ARRAY[1..7,8..19 ] 	OF REAL ;(*历史每天白班每小时产量*)
	(*夜班*)
	NightCountTotalHistory		:ARRAY[1..7 ] 	OF REAL ;
	HMI_NightOkCountHistory		:ARRAY[1..7 ] 	OF REAL ;
	HMI_NightNgCountHistory		:ARRAY[1..7 ] 	OF REAL ;
	HMI_NightQualifiedHistory	:ARRAY[1..7 ] 	OF REAL ;
	NightRunTimeTotalHistory	:ARRAY[1..7 ] 	OF REAL ;
	NightWaitTimeTotalHistory	:ARRAY[1..7 ] 	OF REAL ;
	NightAlarmTimeTotalHistory	:ARRAY[1..7 ] 	OF REAL ;
	NgPerHourNightCountHistory	:ARRAY[1..7,1..30 ] 	OF REAL ;
	HourTimeNightCountHistory	:ARRAY[1..7,0..23] 	OF REAL ;
	(*历史数据变量汇总1-7天*)


(**********************************生产统计数据********************************************)
	DayRunTime_min:ARRAY[8..19] 	OF REAL;	(*白班每小时运行时间*)
	NightRunTime_min:ARRAY[0..23] 	OF REAL;	(*夜班每小时运行时间*)
	AllDayRunTime_min: REAL;	(*白班总运行时间*)
	AllNightRunTime_min: REAL;	(*夜班总运行时间*)

	DayWaitTime_min:ARRAY[8..19] 	OF REAL;	(*白班待料每小时时间*)
	NightWaitTime_min:ARRAY[0..23] 	OF REAL;	(*夜班待料每小时时间*)
	AllDayWaitTime_min: REAL;(*白班总待料时间*)
	AllNightWaitTime_min: REAL;(*夜班总待料时间*)

	DayAlmTime_min:ARRAY[8..19] 	OF REAL;	(*白班每小时报警时间*)
	NightAlmTime_min:ARRAY[0..23] OF REAL;	(*夜班每小时报警时间*)
	AllDayAlmTime_min: REAL;	(*白班总报警时间*)
	AllNightAlmTime_min: REAL;	(*夜班总报警时间*)

	DayBlockTime_min:ARRAY[0..23] 	OF REAL;(*白班每小时堵料时间*)
	NightBlockTime_min:ARRAY[0..23] 	OF REAL;(*夜班每小时堵料时间*)
	AllDayBlockTime_min: REAL;(*白班总堵料时间*)
	AllNightBlockTime_min: REAL;(*夜班总堵料时间*)
	
	HMINgClassCount_Day:ARRAY[1..30,0..23] 	OF REAL;(*白班每种NG类型每小时统计 ,,,NG类型，小时*)
	HMINgClassCount_Night:ARRAY[1..30,0..23] 	OF REAL;(*夜班每种NG类型每小时统计 ,,,NG类型，小时*)
	
	
	

	HisDayRunTime_min	:ARRAY[1..7,8..19 ] OF REAL ; (*历史白班每小时运行时间*)
	HisNightRunTime_min	:ARRAY[1..7,0..23 ] OF REAL ; (*历史夜班每小时运行时间*)
	HisAllDayRunTime_min:ARRAY[1..7] OF REAL ;	(*历史白班总运行时间*)
	HisAllNightRunTime_min:ARRAY[1..7 ] OF REAL ;	(*历史夜班总运行时间*)

	HisDayWaitTime_min	:ARRAY[1..7,8..19 ] OF REAL ; (*历史白班每小时待料时间*)
	HisNightWaitTime_min:ARRAY[1..7,0..23 ] OF REAL ; (*历史夜班每小时待料时间*)
	HisAllDayWaitTime_min:ARRAY[1..7] OF REAL ;	(*历史白班总待料时间*)
	HisAllNightWaitTime_min:ARRAY[1..7 ] OF REAL ;	(*历史夜班总待料时间*)

	HisDayAlmTime_min	:ARRAY[1..7,8..19 ] OF REAL ; (*历史白班每小时报警时间*)
	HisNightAlmTime_min	:ARRAY[1..7,0..23 ] OF REAL ; (*历史夜班每小时报警时间*)
	HisAllDayAlmTime_min:ARRAY[1..7] OF REAL ;	(*历史白班总报警时间*)
	HisAllNightAlmTime_min:ARRAY[1..7 ] OF REAL ;(*历史夜班总报警时间*)

	HisHMINgClassCount_Day:ARRAY[1..30,0..23,1..7] 	OF REAL;(*历史白班每种NG类型每小时统计,,,NG类型，小时，天*)
	HisHMINgClassCount_Night:ARRAY[1..30,0..23,1..7] 	OF REAL;(*历史夜班每种NG类型每小时统计,,,NG类型，小时，天*)

END_STRUCT
END_TYPE

// ---- P2DUTs/38_User1/P2_AxiseNo.TcDUT
TYPE P2_AxiseNo ://伺服轴号、虚轴号
STRUCT
	AxisName:ST_AxisName;//伺服轴号
	VirAxisName:ST_VirAxisName;//虚轴号
END_STRUCT
END_TYPE

// ---- P2DUTs/38_User1/P2_TableNo.TcDUT
TYPE P2_TableNo :           //凸轮表
STRUCT
	  M_GMDanserMove_L	              :UINT;	//  隔膜摆臂左凸轮
      M_GMDanserMove_R	              :UINT;	//  隔膜摆臂左凸轮
	  M_GMWind_L	                          :UINT;	//  隔膜放卷左凸轮
	  M_GMWind2_L	                          :UINT;	//  隔膜放卷左凸轮
      M_GMWind_R	                      :UINT;	//  隔膜放卷右凸轮
	  M_GMWind2_R	                      :UINT;	//  隔膜放卷右凸轮
	  M_GMBuffer_L	                      :UINT;	//  隔膜缓存左凸轮
	   M_GMBuffer2_L	                      :UINT;	//  隔膜缓存左凸轮
      M_GMBuffer_R	                      :UINT;	//  隔膜缓存右凸轮
	   M_GMBuffer2_R	                      :UINT;	//  隔膜缓存右凸轮
	  M_GMLengthCalculate_L	           :UINT;	//  隔膜长度计算左凸轮
	  M_GMLengthCalculate2_L	           :UINT;	//  隔膜长度计算左凸轮
      M_GMLengthCalculate_R	           :UINT;	//  隔膜长度计算右凸轮
	   M_GMLengthCalculate2_R	           :UINT;	//  隔膜长度计算右凸轮
      M_GMVir_L	                               :UINT;	//  隔膜虚轴左凸轮


      M_AnCarryingLine                     :UINT; //		正极送片搬运平移
      M_AnCarryingUpDown               :UINT; //		正极送片搬运升降取片
	  M_AnCarryingUpDown1               :UINT; //	正极送片搬运升降放片
	   M_AnCarryingUpDown3               :UINT; //	正极送片搬运升降避让
      M_AnCarryingWhirling               :UINT; //		正极送片搬运旋转
      M_AnDTCarryingLine                  :UINT; //		正极叠台搬运平移
      M_AnDTCarryingUpDown            :UINT; //		正极叠台搬运升降取片
	  M_AnDTCarryingUpDown1            :UINT; //		正极叠台搬运升降放片	
	  M_AnDTCarryingUpDown3            :UINT; //		正极叠台搬运升降避让
	  
      M_CaCarryingLine1                     :UINT; //		负极送片搬运1平移
      M_CaCarryingUpDown1               :UINT; //    负极送片搬运1放片升降
	  M_CaCarryingUpDown1_1               :UINT; //    负极送片搬运1取片升降
	
      M_CaCarryingWhirling1               :UINT; //		负极送片搬运1旋转
      M_CaCarryingLine2                     :UINT; //		负极送片搬运2平移
      M_CaCarryingUpDown2              :UINT; //		负极送片搬运2升降取片
	  M_CaCarryingUpDown2_1              :UINT; //		负极送片搬运2升降放片
	  M_CaCarryingUpDown2_3              :UINT; //		负极送片搬运2升降避让
      M_CaBelt                                   :UINT; //		负极送片皮带
      M_CaDTCarryingLine                  :UINT; //		负极叠台搬运平移
      M_CaDTCarryingUpDown            :UINT; //		负极叠台搬运升降取片
	  M_CaDTCarryingUpDown1            :UINT; //		负极叠台搬运升降放片
	  M_CaDTCarryingUpDown3            :UINT; //		负极叠台搬运升降放片
     M_DTUpDown	                             :UINT;	//	叠台升降
     M_LeftYDLine                                :UINT;	//	左压刀开合
     M_LeftYDUpDown                         :UINT;	//	左压刀升降
     M_RightYDLine	                            :UINT;	//	右压刀开合
     M_RightYDUpDown                       :UINT;	//	右压刀升降

	 M_TailCurlLine                        	     :UINT;	//	尾卷平移
	 M_TailCurlUpDown	                     :UINT;	//	尾卷升降
	 
     M_LeftYDLine2                           :UINT;	//	左压刀开合2
     M_LeftYDUpDown2                         :UINT;	//	左压刀升降2
     M_RightYDLine2	                        :UINT;	//	右压刀开合2
     M_RightYDUpDown2                       :UINT;	//	右压刀升降2	 

END_STRUCT
END_TYPE

// ---- P2DUTs/38_User1/Parameters.TcDUT
TYPE  Parameters :
STRUCT
	(*
	An_Quantity:UINT;//正极设定极片数		
	Ca_Quantity:UINT;//负极设定极片数
	Ca_betlCount:word_bool;//负极极片级存流水线记录极片数
	
	Stickersettings:word_bool;//贴胶设置需要贴的胶道数
	StickerDone:word_bool;//已贴胶的道数
	*)

    stDT_date:parDT_date;//叠台设定断电保持参数

    Mechaical:  parMechanical;  //机械参数
	
	stWJ_date:parTailCurl_date;//尾卷设定参数

   
    iStationNO:    INT;  //叠片站好    1:1#叠片     2:1#叠片     3:1#叠片   
   
  	Code:     ParCode;   //二维码参数
	iModeEN             : IModeEN;//功能屏蔽

END_STRUCT
END_TYPE

// ---- P2DUTs/38_User1/sMC_CAM_REF.TcDUT
TYPE sMC_CAM_REF :
STRUCT
	Distance:REAL;
	Phase:REAL;
END_STRUCT
END_TYPE

// ---- P2DUTs/38_User1/System_Control.TcDUT
TYPE System_Control :
STRUCT
	btn:ST_SystemButton;//系统按钮
	se:System_Senser;//系统信号
END_STRUCT
END_TYPE

// ---- P2DUTs/38_User1/User1_Par.TcDUT
TYPE User1_Par :
STRUCT
 	// iTargetTorque	                 	:ARRAY[1..3]OF INT:= [3(-50)];			                     (*单位为0.1%*)
     iTest                                   :INT;

     parFilterAD              :ARRAY[1..MaxAINo] OF ST_ParFilterAD;
     parDA                     :ARRAY[1..44] OF INT;   //模拟量输出
	HMI_Version					:STRING:='V20221208';//触摸屏版本号
	PLC_Version					:STRING:='V20221208';//PLC版本号
    bSyncMode:INT:=1;//0=不同步启动叠台主轴，1=同时启动叠台主轴






END_STRUCT
END_TYPE

// ---- P2DUTs/39User2/conAn_date.TcDUT
TYPE conAn_date ://正极取片
STRUCT
	
	An_GohomeHMI:BOOL;//正极回原点启动
	An_GohomeDone:BOOL;//正极回原点完成
	An_Quantited:UINT;//正极已叠数量
	An_KDQuantited:UINT;//正极空叠隔膜已叠片数
	An_EmptyRunKDQuantited:UINT;//正极空跑模式空叠隔膜已叠层数
	//An_KDQuantited:UINT;//正极空叠隔膜已叠片数
	An_CarryingFalg:BOOL;//正极搬运吸盘有无料标记
	An_QuLiaoOK:BOOL;//正极取流水线极片允许
	An_deviationFalg:BOOL;//正极纠偏平台有无料标记
	An_DPCarryingFalg:BOOL;//正极叠台搬运 吸盘有无料标记
	An_DPRequest:BOOL;//正极叠片请求
	An_BlueflagingKDSet:UINT;//正极接带空叠隔膜设定片数
	An_YellowmarkKDSet:UINT;//正极极色标空叠隔膜设定片数
	An_Blueflaging_TF:UINT;//正极蓝胶标记空叠层数	
	
	
	//An_deviationCCDOK:BOOL;//正极纠偏平台拍照OK
	//An_deviationCCDNG:BOOL;//正极纠偏平台拍照NG
	An_CCDStart:BOOL;//正极CCD拍照启动
	An_deviationCCDDone:BOOL;//正极CCD拍照完成
	
	An_deviationFPOK:BOOL;//正极纠偏平台允许放极片
	An_deviationDPOK:BOOL;//正极纠偏平台允许取极片
	An_deviationDone:BOOL;//正极纠偏平台纠偏完成
	An_MainBeltOK:BOOL;//正极流水线主分料皮带允许取极片
	An_MainBelting:BOOL;//正极流水线主分料皮带取极片中
	AN_AxisCarrying:BOOL;//正极各轴正在运行到初始位中
	AN_BeltDone:BOOL;//正极取主分料流水线极片完成
	AN_BeltSafe:BOOL;//正极取主分料流水线极片安全位
	GetPiceReady:BOOL;//正极准备好取分段流水线上的极片
	JumpPiceReady:BOOL;//正极放弃取分段流水线上的极片	
	bAn_PoleHave:BOOL;//正极取料位无片
	
	An_StandbyStep:ARRAY[0..9] OF UINT;//正极备极片程序步
	CarryingSafepos:ARRAY[0..9] OF BOOL;//正极搬动轴在安全位置指示
	Error: ARRAY[0..80] OF BOOL;//报警
	Error_tips	:ARRAY[0..60] OF BOOL;//报警提示
	
	RectifydevStart:BOOL; //纠偏启动
	RectifydevDone:BOOL; //纠偏完成
	
	//CCD_X1:REAL; //纠偏平台X1的纠偏量
	//CCD_X2:REAL;//纠偏平台X2的纠偏量
	//CCD_Y:REAL;//纠偏平台Y的纠偏量	
	
	DemarcateStart:BOOL; //标定启动	
	DemarcateDone:BOOL; //CCD标定完成
	Demarcateing:BOOL;//CCD标定中
	
	CreateCamStart:BOOL;//正极取片凸轮创建
	CreateCamDone:BOOL;//正极取片凸轮创建完成
	
	bAnCCD_TestDo:BOOL;//正极CCD测试开始
	iAnCCD_PhotoCT:INT;//正极拍照取图时间
	iAnCCD_RectifyCT:INT;//正极纠偏时间	
	An_CCD_amount :int;//正极连续NG计数
	An_DTqr :BOOL;//正极极片掉片人工确认按钮
	An_Rectifydev_CQ :BOOL;//正极纠偏平台除尘
	An_Rectifydev_CS :INT;//纠偏计数
	
	An_Rectifydev_PB :BOOL;//二次纠偏屏蔽 OFF：屏蔽二次纠偏
	An_VacuumErrorNG :BOOL;//正极抛真空NG料标志
	//新增，首层隔膜
	An_FirstFoldCnt:INT;//正极首层隔膜已叠次数
	An_FirstFoldSet:INT:=1;//正极首层隔膜设定次数
		//20240414WCZ
	RectifyTryStart:BOOL;//CCD重复精度测试启动
	SuckerTestStart:BOOL;//吸盘重复精度测试启动
END_STRUCT
END_TYPE

// ---- P2DUTs/39User2/conCa_date.TcDUT
TYPE conCa_date ://负极取片
STRUCT
	
	Ca_GohomeHMI:BOOL;//负极回原点启动
	Ca_GohomeDone:BOOL;//负极回原点完成
	
	Ca_BeltGohomeHMI:BOOL;//负极回原点启动
	Ca_BeltGohomeDone:BOOL;//负极回原点完成
	
